C01815=1042.872,189.245,401.631,170.706,39.052,157.377
C01816=1042.879,189.530,401.603,170.709,39.053,157.377
C01817=1042.886,189.814,401.575,170.712,39.055,157.378
C01818=1042.893,190.099,401.548,170.715,39.057,157.378
C01819=1042.899,190.347,401.523,170.718,39.058,157.378
C01820=1042.905,190.596,401.499,170.720,39.060,157.379
C01821=1042.911,190.845,401.475,170.723,39.061,157.379
C01822=1042.918,191.094,401.450,170.726,39.062,157.380
C01823=1042.923,191.342,401.426,170.728,39.064,157.380
C01824=1042.929,191.591,401.402,170.731,39.065,157.380
C01825=1042.935,191.839,401.377,170.734,39.067,157.381
C01826=1042.941,192.089,401.353,170.737,39.068,157.381
C01827=1042.948,192.338,401.329,170.739,39.070,157.381
C01828=1042.953,192.586,401.304,170.742,39.071,157.382
C01829=1042.960,192.835,401.280,170.745,39.072,157.382
C01830=1042.965,193.083,401.255,170.747,39.074,157.383
C01831=1042.972,193.332,401.231,170.750,39.075,157.383
C01832=1042.978,193.581,401.207,170.753,39.077,157.383
C01833=1042.984,193.829,401.182,170.755,39.078,157.384
C01834=1042.990,194.078,401.158,170.759,39.080,157.384
C01835=1042.997,194.327,401.134,170.761,39.081,157.384
C01836=1043.002,194.575,401.109,170.763,39.082,157.385
C01837=1043.009,194.824,401.085,170.767,39.084,157.385
C01838=1043.015,195.074,401.060,170.769,39.085,157.385
C01839=1043.021,195.322,401.035,170.772,39.087,157.386
C01840=1043.027,195.571,401.011,170.775,39.088,157.386
C01841=1043.033,195.819,400.986,170.778,39.089,157.387
C01842=1043.040,196.068,400.962,170.780,39.091,157.387
C01843=1043.045,196.317,400.937,170.783,39.093,157.387
C01844=1043.052,196.565,400.913,170.786,39.094,157.388
C01845=1043.058,196.814,400.888,170.789,39.096,157.388
C01846=1043.064,197.063,400.863,170.792,39.097,157.389
C01847=1043.070,197.311,400.839,170.794,39.098,157.389
C01848=1043.076,197.560,400.814,170.798,39.100,157.389
C01849=1043.083,197.809,400.790,170.800,39.101,157.390
C01850=1043.089,198.058,400.765,170.802,39.103,157.390
C01851=1043.096,198.307,400.740,170.806,39.105,157.391
C01852=1043.101,198.555,400.716,170.808,39.106,157.391
C01853=1043.107,198.804,400.691,170.811,39.107,157.391
C01854=1043.114,199.053,400.667,170.814,39.109,157.392
C01855=1043.120,199.302,400.641,170.817,39.110,157.392
C01856=1043.127,199.550,400.617,170.819,39.112,157.392
C01857=1043.132,199.798,400.592,170.823,39.113,157.393
C01858=1043.139,200.047,400.568,170.825,39.114,157.393
C01859=1043.145,200.296,400.543,170.828,39.116,157.394
C01860=1043.152,200.545,400.518,170.831,39.118,157.394
C01861=1043.158,200.794,400.494,170.834,39.119,157.394
C01862=1043.164,201.042,400.468,170.836,39.121,157.395
C01863=1043.170,201.290,400.443,170.840,39.122,157.395
C01864=1043.176,201.540,400.419,170.842,39.124,157.396
C01865=1043.183,201.788,400.394,170.846,39.126,157.396
C01866=1043.189,202.037,400.369,170.848,39.127,157.396
C01867=1043.195,202.285,400.343,170.850,39.129,157.397
C01868=1043.201,202.535,400.319,170.854,39.130,157.397
C01869=1043.207,202.783,400.294,170.856,39.132,157.398
C01870=1043.213,203.031,400.268,170.860,39.133,157.398
C01871=1043.219,203.280,400.243,170.862,39.135,157.398
C01872=1043.225,203.529,400.218,170.865,39.137,157.399
C01873=1043.231,203.778,400.193,170.868,39.138,157.399
C01874=1043.237,204.027,400.168,170.871,39.140,157.400
C01875=1043.243,204.275,400.143,170.873,39.142,157.400
C01876=1043.249,204.523,400.117,170.877,39.143,157.401
C01877=1043.255,204.772,400.092,170.879,39.145,157.401
C01878=1043.262,205.021,400.068,170.883,39.147,157.401
C01879=1043.288,206.072,399.961,171.152,39.248,157.431
C01880=1043.296,206.361,399.930,171.154,39.251,157.431
C01881=1043.303,206.650,399.900,171.156,39.254,157.432
C01882=1043.311,206.938,399.870,171.159,39.257,157.432
C01883=1043.319,207.228,399.839,171.162,39.260,157.433
C01884=1043.326,207.476,399.813,171.164,39.262,157.434
C01885=1043.332,207.725,399.786,171.166,39.264,157.434
C01886=1043.339,207.973,399.759,171.168,39.267,157.435
C01887=1043.346,208.222,399.733,171.170,39.269,157.435
C01888=1043.352,208.470,399.707,171.172,39.271,157.436
C01889=1043.359,208.719,399.680,171.175,39.273,157.436
C01890=1043.365,208.967,399.654,171.177,39.276,157.437
C01891=1043.372,209.215,399.628,171.179,39.279,157.438
C01892=1043.379,209.465,399.601,171.181,39.281,157.438
C01893=1043.385,209.713,399.574,171.183,39.283,157.439
C01894=1043.392,209.962,399.547,171.186,39.286,157.439
C01895=1043.398,210.210,399.521,171.187,39.288,157.440
C01896=1043.405,210.458,399.495,171.190,39.290,157.440
C01897=1043.411,210.707,399.468,171.191,39.293,157.441
C01898=1043.418,210.956,399.442,171.194,39.295,157.442
C01899=1043.425,211.203,399.415,171.196,39.297,157.442
C01900=1043.431,211.452,399.388,171.198,39.300,157.443
C01901=1043.438,211.701,399.362,171.200,39.302,157.443
C01902=1043.444,211.949,399.335,171.203,39.304,157.444
C01903=1043.451,212.198,399.309,171.205,39.307,157.445
C01904=1043.457,212.446,399.282,171.207,39.310,157.445
C01905=1043.464,212.694,399.255,171.209,39.312,157.446
C01906=1043.470,212.943,399.228,171.211,39.314,157.446
C01907=1043.477,213.192,399.202,171.214,39.317,157.447
C01908=1043.484,213.441,399.175,171.215,39.319,157.447
C01909=1043.490,213.688,399.147,171.218,39.321,157.448
C01910=1043.497,213.937,399.121,171.220,39.324,157.448
C01911=1043.503,214.185,399.094,171.222,39.327,157.449
C01912=1043.510,214.434,399.068,171.225,39.329,157.450
C01913=1043.516,214.683,399.040,171.227,39.331,157.450
C01914=1043.523,214.931,399.014,171.229,39.334,157.451
C01915=1043.529,215.180,398.987,171.231,39.336,157.451
C01916=1043.537,215.428,398.960,171.234,39.338,157.452
C01917=1043.543,215.676,398.933,171.235,39.341,157.452
C01918=1043.549,215.925,398.906,171.238,39.343,157.453
C01919=1043.556,216.173,398.879,171.240,39.345,157.454
C01920=1043.562,216.422,398.853,171.242,39.348,157.454
C01921=1043.569,216.671,398.826,171.244,39.350,157.455
C01922=1043.576,216.919,398.798,171.247,39.352,157.455
C01923=1043.582,217.167,398.772,171.248,39.355,157.456
C01924=1043.589,217.416,398.745,171.251,39.357,157.456
C01925=1043.595,217.665,398.718,171.254,39.360,157.457
C01926=1043.602,217.913,398.692,171.256,39.362,157.458
C01927=1043.609,218.161,398.664,171.258,39.364,157.458
C01928=1043.616,218.410,398.637,171.260,39.367,157.459
C01929=1043.622,218.658,398.611,171.263,39.369,157.459
C01930=1043.628,218.907,398.583,171.264,39.371,157.460
C01931=1043.635,219.155,398.557,171.267,39.374,157.460
C01932=1043.642,219.404,398.529,171.269,39.376,157.461
C01933=1043.649,219.652,398.503,171.272,39.378,157.461
C01934=1043.655,219.900,398.475,171.274,39.381,157.462
C01935=1043.662,220.149,398.448,171.276,39.383,157.463
C01936=1043.670,220.443,398.416,171.279,39.386,157.463
C01937=1043.678,220.737,398.384,171.281,39.389,157.464
C01938=1043.685,221.032,398.351,171.284,39.391,157.465
C01939=1043.692,221.326,398.320,171.287,39.394,157.465
C01940=1043.699,221.574,398.292,171.289,39.396,157.466
C01941=1043.706,221.823,398.264,171.292,39.399,157.467
C01942=1043.712,222.072,398.237,171.293,39.402,157.467
C01943=1043.718,222.320,398.210,171.296,39.404,157.468
C01944=1043.726,222.568,398.183,171.299,39.406,157.468
C01945=1043.732,222.817,398.156,171.301,39.408,157.469
C01946=1043.739,223.065,398.128,171.304,39.411,157.469
C01947=1043.745,223.313,398.101,171.305,39.413,157.470
C01948=1043.751,223.562,398.074,171.308,39.415,157.470
C01949=1043.758,223.810,398.046,171.310,39.418,157.471
C01950=1043.765,224.059,398.018,171.313,39.420,157.472
C01951=1043.771,224.308,397.991,171.314,39.422,157.472
C01952=1043.778,224.555,397.964,171.317,39.425,157.473
C01953=1043.784,224.804,397.937,171.320,39.427,157.473
C01954=1043.791,225.052,397.909,171.322,39.430,157.474
C01955=1043.797,225.301,397.882,171.324,39.432,157.474
C01956=1043.804,225.550,397.854,171.326,39.434,157.475
C01957=1043.810,225.798,397.827,171.329,39.437,157.476
C01958=1043.817,226.046,397.799,171.331,39.439,157.476
C01959=1043.824,226.294,397.771,171.334,39.441,157.477
C01960=1043.831,226.543,397.745,171.336,39.444,157.477
C01961=1043.837,226.792,397.717,171.338,39.446,157.478
C01962=1043.844,227.040,397.689,171.340,39.448,157.478
C01963=1043.851,227.288,397.662,171.343,39.450,157.479
C01964=1043.857,227.536,397.634,171.346,39.453,157.480
C01965=1043.864,227.785,397.607,171.348,39.455,157.480
C01966=1043.870,228.034,397.580,171.350,39.457,157.481
C01967=1043.877,228.282,397.552,171.352,39.460,157.481
C01968=1043.883,228.531,397.524,171.355,39.462,157.482
C01969=1043.890,228.779,397.496,171.357,39.464,157.482
C01970=1043.897,229.027,397.469,171.360,39.467,157.483
C01971=1043.903,229.276,397.441,171.363,39.469,157.484
C01972=1043.909,229.524,397.414,171.364,39.472,157.484
C01973=1043.916,229.772,397.386,171.367,39.474,157.485
C01974=1043.923,230.021,397.358,171.369,39.476,157.485
C01975=1043.929,230.269,397.330,171.372,39.479,157.486
C01976=1043.936,230.517,397.303,171.374,39.481,157.486
C01977=1043.943,230.766,397.275,171.377,39.483,157.487
C01978=1043.949,231.015,397.247,171.379,39.485,157.488
C01979=1043.955,231.263,397.219,171.381,39.488,157.488
C01980=1043.962,231.512,397.191,171.384,39.491,157.489
C01981=1043.968,231.759,397.164,171.386,39.493,157.489
C01982=1043.975,232.008,397.136,171.389,39.495,157.490
C01983=1043.982,232.255,397.108,171.391,39.498,157.491
C01984=1043.989,232.504,397.080,171.394,39.500,157.491
C01985=1043.994,232.753,397.052,171.396,39.502,157.492
C01986=1044.001,233.001,397.024,171.398,39.504,157.492
C01987=1044.008,233.250,396.996,171.401,39.507,157.493
C01988=1044.015,233.498,396.968,171.403,39.510,157.494
C01989=1044.020,233.747,396.940,171.406,39.512,157.494
C01990=1044.027,233.995,396.912,171.408,39.514,157.495
C01991=1044.034,234.243,396.884,171.411,39.516,157.495
C01992=1044.041,234.530,396.852,171.414,39.519,157.496
C01993=1044.049,234.817,396.819,171.416,39.522,157.496
C01994=1044.056,235.103,396.787,171.419,39.525,157.497
C01995=1044.064,235.390,396.754,171.423,39.527,157.498
C01996=1044.071,235.639,396.727,171.424,39.530,157.498
C01997=1044.077,235.887,396.698,171.427,39.532,157.499
C01998=1044.084,236.135,396.670,171.429,39.534,157.500
C01999=1044.090,236.384,396.642,171.432,39.537,157.500
C02000=1044.096,236.632,396.614,171.434,39.539,157.501
C02001=1044.103,236.880,396.585,171.437,39.542,157.501
C02002=1044.110,237.129,396.558,171.440,39.544,157.502
C02003=1044.117,237.377,396.530,171.442,39.546,157.503
C02004=1044.123,237.625,396.501,171.445,39.548,157.503
C02005=1044.130,237.874,396.473,171.447,39.551,157.504
C02006=1044.137,238.122,396.445,171.450,39.553,157.504
C02007=1044.143,238.370,396.416,171.452,39.555,157.505
C02008=1044.149,238.619,396.389,171.455,39.558,157.505
C02009=1044.156,238.867,396.360,171.458,39.560,157.506
C02010=1044.162,239.115,396.332,171.460,39.563,157.507
C02011=1044.169,239.363,396.304,171.463,39.565,157.507
C02012=1044.176,239.612,396.276,171.465,39.567,157.508
C02013=1044.183,239.860,396.246,171.467,39.570,157.508
C02014=1044.189,240.109,396.219,171.469,39.572,157.509
C02015=1044.195,240.358,396.190,171.472,39.574,157.510
C02016=1044.202,240.605,396.162,171.475,39.576,157.510
C02017=1044.209,240.854,396.134,171.477,39.579,157.511
C02018=1044.215,241.102,396.105,171.480,39.581,157.511
C02019=1044.222,241.350,396.077,171.482,39.583,157.512
C02020=1044.228,241.599,396.048,171.485,39.586,157.513
C02021=1044.235,241.846,396.020,171.488,39.588,157.513
C02022=1044.241,242.095,395.992,171.490,39.591,157.514
C02023=1044.248,242.343,395.963,171.493,39.593,157.514
C02024=1044.255,242.592,395.934,171.495,39.595,157.515
C02025=1044.261,242.841,395.905,171.498,39.598,157.516
C02026=1044.268,243.088,395.877,171.501,39.600,157.516
C02027=1044.274,243.336,395.848,171.503,39.603,157.517
C02028=1044.281,243.585,395.820,171.506,39.605,157.517
C02029=1044.287,243.833,395.791,171.508,39.607,157.518
C02030=1044.293,244.081,395.762,171.511,39.610,157.519
C02031=1044.300,244.330,395.734,171.513,39.612,157.519
C02032=1044.307,244.578,395.705,171.516,39.615,157.520
C02033=1044.314,244.826,395.677,171.519,39.617,157.520
C02034=1044.320,245.074,395.647,171.521,39.619,157.521
C02035=1044.326,245.323,395.619,171.524,39.621,157.521
C02036=1044.333,245.571,395.591,171.526,39.624,157.522
C02037=1044.339,245.819,395.562,171.529,39.626,157.523
C02038=1044.346,246.067,395.533,171.532,39.629,157.523
C02039=1044.352,246.315,395.504,171.534,39.632,157.524
C02040=1044.359,246.564,395.474,171.537,39.634,157.525
C02041=1044.365,246.813,395.446,171.539,39.636,157.525
C02042=1044.371,247.061,395.417,171.542,39.638,157.526
C02043=1044.378,247.309,395.388,171.545,39.641,157.526
C02044=1044.384,247.557,395.359,171.547,39.643,157.527
C02045=1044.390,247.805,395.330,171.551,39.646,157.528
C02046=1044.397,248.054,395.301,171.553,39.648,157.528
C02047=1044.403,248.302,395.272,171.556,39.651,157.529
C02048=1044.410,248.583,395.239,171.559,39.654,157.530
C02049=1044.418,248.864,395.206,171.561,39.656,157.530
C02050=1044.426,249.145,395.174,171.565,39.659,157.531
C02051=1044.433,249.425,395.141,171.568,39.662,157.532
C02052=1044.440,249.674,395.111,171.570,39.664,157.532
C02053=1044.446,249.922,395.082,171.573,39.667,157.533
C02054=1044.452,250.170,395.053,171.576,39.669,157.533
C02055=1044.458,250.419,395.024,171.578,39.671,157.534
C02056=1044.465,250.667,394.995,171.581,39.673,157.535
C02057=1044.471,250.916,394.966,171.584,39.676,157.535
C02058=1044.478,251.163,394.937,171.586,39.679,157.536
C02059=1044.485,251.411,394.908,171.590,39.681,157.536
C02060=1044.491,251.660,394.879,171.592,39.683,157.537
C02061=1044.498,251.908,394.850,171.595,39.686,157.538
C02062=1044.504,252.157,394.821,171.598,39.688,157.538
C02063=1044.511,252.404,394.791,171.600,39.690,157.539
C02064=1044.517,252.653,394.762,171.603,39.693,157.539
C02065=1044.524,252.901,394.733,171.605,39.695,157.540
C02066=1044.530,253.149,394.704,171.608,39.698,157.541
C02067=1044.537,253.398,394.674,171.611,39.700,157.541
C02068=1044.544,253.646,394.646,171.614,39.702,157.542
C02069=1044.550,253.893,394.616,171.617,39.705,157.543
C02070=1044.557,254.142,394.587,171.619,39.707,157.543
C02071=1044.563,254.390,394.557,171.622,39.709,157.544
C02072=1044.570,254.638,394.528,171.625,39.712,157.544
C02073=1044.577,254.887,394.498,171.627,39.715,157.545
C02074=1044.583,255.135,394.469,171.630,39.717,157.546
C02075=1044.589,255.383,394.440,171.633,39.719,157.546
C02076=1044.596,255.632,394.411,171.636,39.721,157.547
C02077=1044.603,255.879,394.381,171.639,39.724,157.547
C02078=1044.610,256.128,394.352,171.641,39.726,157.548
C02079=1044.616,256.376,394.323,171.644,39.729,157.549
C02080=1044.623,256.623,394.293,171.647,39.731,157.549
C02081=1044.630,256.872,394.264,171.650,39.733,157.550
C02082=1044.636,257.120,394.235,171.653,39.736,157.551
C02083=1044.643,257.369,394.205,171.655,39.738,157.551
C02084=1044.650,257.617,394.176,171.658,39.740,157.552
C02085=1044.656,257.864,394.146,171.661,39.743,157.552
C02086=1044.663,258.113,394.117,171.664,39.745,157.553
C02087=1044.669,258.361,394.088,171.667,39.748,157.554
C02088=1044.676,258.609,394.058,171.669,39.750,157.554
C02089=1044.683,258.858,394.029,171.672,39.752,157.555
C02090=1044.690,259.106,393.998,171.676,39.755,157.556
C02091=1044.696,259.354,393.969,171.678,39.757,157.556
C02092=1044.703,259.602,393.939,171.681,39.759,157.557
C02093=1044.709,259.850,393.910,171.683,39.762,157.557
C02094=1044.717,260.098,393.880,171.686,39.764,157.558
C02095=1044.723,260.347,393.851,171.690,39.767,157.559
C02096=1044.730,260.595,393.821,171.692,39.769,157.559
C02097=1044.736,260.843,393.792,171.695,39.771,157.560
C02098=1044.743,261.091,393.762,171.698,39.773,157.560
C02099=1044.750,261.339,393.733,171.701,39.776,157.561
C02100=1044.757,261.588,393.703,171.704,39.778,157.562
C02101=1044.763,261.836,393.674,171.706,39.781,157.562
C02102=1044.771,262.084,393.644,171.709,39.783,157.563
C02103=1044.778,262.332,393.614,171.713,39.785,157.563
C02104=1044.785,262.611,393.581,171.715,39.788,157.564
C02105=1044.792,262.891,393.547,171.719,39.791,157.565
C02106=1044.800,263.171,393.513,171.722,39.793,157.566
C02107=1044.806,263.450,393.480,171.726,39.796,157.566
C02108=1044.814,263.698,393.450,171.728,39.799,157.567
C02109=1044.819,263.946,393.419,171.731,39.801,157.568
C02110=1044.827,264.194,393.389,171.734,39.803,157.568
C02111=1044.833,264.442,393.359,171.737,39.806,157.569
C02112=1044.839,264.691,393.329,171.740,39.808,157.569
C02113=1044.846,264.939,393.299,171.742,39.811,157.570
C02114=1044.853,265.187,393.269,171.746,39.813,157.571
C02115=1044.859,265.435,393.239,171.749,39.816,157.571
C02116=1044.866,265.683,393.209,171.751,39.819,157.572
C02117=1044.873,265.931,393.179,171.755,39.821,157.573
C02118=1044.879,266.179,393.149,171.758,39.824,157.573
C02119=1044.886,266.428,393.119,171.760,39.826,157.574
C02120=1044.893,266.676,393.089,171.763,39.828,157.575
C02121=1044.899,266.924,393.059,171.767,39.831,157.575
C02122=1044.906,267.172,393.029,171.769,39.833,157.576
C02123=1044.912,267.419,392.999,171.772,39.836,157.577
C02124=1044.919,267.668,392.968,171.776,39.838,157.577
C02125=1044.926,267.916,392.938,171.778,39.841,157.578
C02126=1044.932,268.164,392.908,171.781,39.843,157.579
C02127=1044.939,268.412,392.877,171.784,39.845,157.579
C02128=1044.945,268.660,392.847,171.787,39.848,157.580
C02129=1044.952,268.908,392.817,171.790,39.850,157.580
C02130=1044.958,269.157,392.786,171.794,39.853,157.581
C02131=1044.965,269.404,392.757,171.796,39.855,157.582
C02132=1044.971,269.653,392.726,171.799,39.858,157.582
C02133=1044.979,269.900,392.695,171.802,39.860,157.583
C02134=1044.985,270.148,392.665,171.805,39.863,157.584
C02135=1044.992,270.396,392.634,171.808,39.865,157.584
C02136=1044.998,270.645,392.604,171.811,39.868,157.585
C02137=1045.005,270.892,392.574,171.814,39.870,157.586
C02138=1045.011,271.141,392.543,171.817,39.873,157.586
C02139=1045.018,271.389,392.513,171.820,39.875,157.587
C02140=1045.024,271.636,392.482,171.823,39.878,157.588
C02141=1045.032,271.884,392.452,171.826,39.880,157.588
C02142=1045.038,272.133,392.421,171.829,39.883,157.589
C02143=1045.044,272.381,392.391,171.832,39.885,157.590
C02144=1045.051,272.628,392.360,171.836,39.888,157.590
C02145=1045.058,272.877,392.329,171.838,39.890,157.591
C02146=1045.063,273.125,392.299,171.841,39.893,157.592
C02147=1045.071,273.373,392.269,171.845,39.895,157.592
C02148=1045.077,273.621,392.237,171.847,39.898,157.593
C02149=1045.084,273.869,392.207,171.850,39.900,157.594
C02150=1045.091,274.116,392.176,171.854,39.903,157.594
C02151=1045.097,274.365,392.146,171.857,39.906,157.595
C02152=1045.103,274.613,392.115,171.860,39.908,157.596
C02153=1045.111,274.861,392.084,171.863,39.911,157.596
C02154=1045.117,275.109,392.054,171.866,39.913,157.597
C02155=1045.123,275.357,392.022,171.869,39.916,157.598
C02156=1045.130,275.605,391.992,171.872,39.918,157.598
C02157=1045.137,275.853,391.961,171.876,39.921,157.599
C02158=1045.143,276.101,391.930,171.878,39.923,157.600
C02159=1045.150,276.349,391.900,171.882,39.926,157.600
C02160=1045.158,276.633,391.864,171.885,39.928,157.601
C02161=1045.165,276.917,391.829,171.889,39.932,157.602
C02162=1045.173,277.201,391.793,171.892,39.934,157.603
C02163=1045.181,277.485,391.758,171.896,39.937,157.603
C02164=1045.187,277.732,391.727,171.899,39.940,157.604
C02165=1045.193,277.981,391.696,171.902,39.942,157.605
C02166=1045.200,278.229,391.665,171.905,39.945,157.606
C02167=1045.207,278.476,391.634,171.908,39.948,157.606
C02168=1045.214,278.725,391.603,171.912,39.950,157.607
C02169=1045.220,278.973,391.572,171.914,39.953,157.608
C02170=1045.227,279.221,391.541,171.918,39.955,157.608
C02171=1045.233,279.468,391.510,171.921,39.958,157.609
C02172=1045.240,279.716,391.479,171.924,39.960,157.610
C02173=1045.246,279.964,391.447,171.927,39.963,157.610
C02174=1045.253,280.213,391.416,171.931,39.965,157.611
C02175=1045.260,280.461,391.385,171.933,39.968,157.612
C02176=1045.266,280.709,391.354,171.937,39.971,157.612
C02177=1045.272,280.956,391.323,171.940,39.974,157.613
C02178=1045.279,281.204,391.292,171.944,39.976,157.614
C02179=1045.286,281.452,391.260,171.946,39.979,157.614
C02180=1045.292,281.700,391.229,171.950,39.981,157.615
C02181=1045.299,281.948,391.198,171.953,39.984,157.616
C02182=1045.306,282.196,391.166,171.956,39.986,157.617
C02183=1045.312,282.444,391.135,171.959,39.989,157.617
C02184=1045.319,282.692,391.103,171.963,39.992,157.618
C02185=1045.326,282.940,391.072,171.966,39.995,157.619
C02186=1045.332,283.187,391.041,171.969,39.997,157.619
C02187=1045.338,283.435,391.010,171.972,40.000,157.620
C02188=1045.345,283.683,390.979,171.976,40.002,157.621
C02189=1045.352,283.931,390.947,171.979,40.005,157.622
C02190=1045.359,284.179,390.916,171.982,40.007,157.622
C02191=1045.365,284.427,390.884,171.985,40.010,157.623
C02192=1045.372,284.675,390.853,171.989,40.013,157.624
C02193=1045.379,284.923,390.821,171.991,40.016,157.624
C02194=1045.386,285.171,390.790,171.995,40.018,157.625
C02195=1045.392,285.419,390.759,171.998,40.020,157.626
C02196=1045.399,285.666,390.727,172.002,40.023,157.626
C02197=1045.406,285.914,390.696,172.005,40.026,157.627
C02198=1045.412,286.162,390.664,172.008,40.028,157.628
C02199=1045.419,286.410,390.633,172.012,40.031,157.629
C02200=1045.426,286.658,390.601,172.014,40.034,157.629
C02201=1045.432,286.906,390.569,172.018,40.036,157.630
C02202=1045.439,287.154,390.537,172.021,40.039,157.631
C02203=1045.446,287.401,390.506,172.025,40.041,157.631
C02204=1045.452,287.649,390.474,172.028,40.044,157.632
C02205=1045.460,287.898,390.443,172.031,40.047,157.633
C02206=1045.466,288.146,390.411,172.035,40.049,157.634
C02207=1045.473,288.393,390.378,172.038,40.052,157.634
C02208=1045.479,288.641,390.347,172.041,40.055,157.635
C02209=1045.486,288.889,390.315,172.045,40.058,157.636
C02210=1045.493,289.137,390.284,172.048,40.060,157.637
C02211=1045.499,289.385,390.251,172.052,40.063,157.637
C02212=1045.506,289.633,390.220,172.054,40.065,157.638
C02213=1045.513,289.881,390.188,172.058,40.068,157.639
C02214=1045.520,290.128,390.156,172.062,40.071,157.639
C02215=1045.526,290.376,390.124,172.065,40.074,157.640
C02216=1045.534,290.672,390.086,172.069,40.077,157.641
C02217=1045.542,290.967,390.048,172.072,40.080,157.642
C02218=1045.550,291.263,390.010,172.077,40.083,157.643
C02219=1045.558,291.559,389.972,172.081,40.087,157.644
C02220=1045.564,291.806,389.939,172.084,40.089,157.644
C02221=1045.571,292.054,389.908,172.088,40.092,157.645
C02222=1045.578,292.302,389.876,172.092,40.095,157.646
C02223=1045.584,292.550,389.844,172.094,40.098,157.647
C02224=1045.591,292.798,389.812,172.098,40.100,157.647
C02225=1045.599,293.045,389.780,172.102,40.103,157.648
C02226=1045.605,293.293,389.747,172.105,40.106,157.649
C02227=1045.612,293.541,389.715,172.108,40.109,157.650
C02228=1045.618,293.789,389.683,172.112,40.111,157.650
C02229=1045.625,294.036,389.651,172.115,40.114,157.651
C02230=1045.632,294.284,389.619,172.119,40.117,157.652
C02231=1045.638,294.532,389.586,172.123,40.119,157.653
C02232=1045.645,294.780,389.555,172.125,40.122,157.653
C02233=1045.651,295.028,389.522,172.129,40.125,157.654
C02234=1045.659,295.275,389.490,172.133,40.128,157.655
C02235=1045.665,295.524,389.457,172.136,40.130,157.656
C02236=1045.672,295.771,389.425,172.139,40.133,157.656
C02237=1045.678,296.019,389.392,172.143,40.136,157.657
C02238=1045.685,296.266,389.360,172.147,40.138,157.658
C02239=1045.691,296.515,389.327,172.150,40.142,157.659
C02240=1045.698,296.762,389.295,172.154,40.145,157.660
C02241=1045.705,297.010,389.262,172.157,40.147,157.660
C02242=1045.711,297.258,389.230,172.160,40.150,157.661
C02243=1045.717,297.505,389.197,172.164,40.153,157.662
C02244=1045.724,297.752,389.165,172.168,40.156,157.663
C02245=1045.731,298.001,389.132,172.171,40.159,157.663
C02246=1045.737,298.248,389.099,172.174,40.161,157.664
C02247=1045.744,298.496,389.066,172.178,40.165,157.665
C02248=1045.750,298.744,389.034,172.181,40.168,157.666
C02249=1045.757,298.992,389.002,172.185,40.170,157.667
C02250=1045.764,299.240,388.969,172.189,40.173,157.667
C02251=1045.770,299.487,388.936,172.193,40.176,157.668
C02252=1045.777,299.736,388.903,172.195,40.179,157.669
C02253=1045.783,299.983,388.870,172.199,40.182,157.670
C02254=1045.790,300.230,388.837,172.203,40.184,157.670
C02255=1045.797,300.477,388.805,172.207,40.188,157.671
C02256=1045.804,300.726,388.772,172.210,40.190,157.672
C02257=1045.810,300.973,388.739,172.213,40.193,157.673
C02258=1045.816,301.221,388.706,172.217,40.196,157.674
C02259=1045.824,301.469,388.674,172.221,40.199,157.674
C02260=1045.830,301.716,388.641,172.224,40.202,157.675
C02261=1045.836,301.964,388.608,172.228,40.205,157.676
C02262=1045.844,302.212,388.574,172.232,40.208,157.677
C02263=1045.850,302.459,388.541,172.235,40.210,157.678
C02264=1045.857,302.708,388.508,172.239,40.214,157.679
C02265=1045.864,302.955,388.476,172.242,40.216,157.679
C02266=1045.870,303.203,388.443,172.246,40.219,157.680
C02267=1045.877,303.450,388.410,172.250,40.222,157.681
C02268=1045.884,303.698,388.377,172.254,40.225,157.682
C02269=1045.891,303.946,388.344,172.257,40.228,157.682
C02270=1045.897,304.194,388.311,172.261,40.231,157.683
C02271=1045.904,304.441,388.277,172.264,40.234,157.684
C02272=1045.913,304.753,388.237,172.269,40.238,157.685
C02273=1045.921,305.065,388.195,172.273,40.241,157.686
C02274=1045.930,305.377,388.153,172.278,40.245,157.687
C02275=1045.939,305.688,388.111,172.283,40.248,157.688
C02276=1045.945,305.937,388.078,172.287,40.252,157.689
C02277=1045.952,306.184,388.045,172.290,40.254,157.690
C02278=1045.959,306.432,388.012,172.294,40.257,157.691
C02279=1045.965,306.679,387.979,172.298,40.260,157.691
C02280=1045.972,306.927,387.945,172.302,40.263,157.692
C02281=1045.979,307.174,387.913,172.306,40.266,157.693
C02282=1045.987,307.422,387.879,172.309,40.269,157.694
C02283=1045.993,307.670,387.846,172.313,40.272,157.695
C02284=1046.000,307.917,387.812,172.317,40.275,157.696
C02285=1046.007,308.166,387.779,172.320,40.278,157.696
C02286=1046.014,308.413,387.746,172.324,40.281,157.697
C02287=1046.020,308.661,387.713,172.328,40.284,157.698
C02288=1046.027,308.908,387.679,172.332,40.287,157.699
C02289=1046.034,309.155,387.645,172.335,40.289,157.700
C02290=1046.042,309.403,387.613,172.339,40.293,157.700
C02291=1046.049,309.650,387.579,172.343,40.295,157.701
C02292=1046.055,309.899,387.546,172.347,40.299,157.702
C02293=1046.063,310.146,387.513,172.351,40.301,157.703
C02294=1046.069,310.393,387.479,172.355,40.305,157.704
C02295=1046.076,310.642,387.446,172.359,40.307,157.705
C02296=1046.083,310.889,387.412,172.363,40.310,157.705
C02297=1046.090,311.136,387.379,172.366,40.313,157.706
C02298=1046.097,311.384,387.345,172.370,40.316,157.707
C02299=1046.104,311.632,387.312,172.374,40.319,157.708
C02300=1046.111,311.880,387.278,172.378,40.322,157.709
C02301=1046.119,312.127,387.245,172.382,40.325,157.710
C02302=1046.126,312.374,387.211,172.386,40.328,157.711
C02303=1046.133,312.623,387.178,172.390,40.331,157.711
C02304=1046.139,312.870,387.144,172.393,40.334,157.712
C02305=1046.146,313.118,387.110,172.397,40.337,157.713
C02306=1046.152,313.366,387.076,172.401,40.341,157.714
C02307=1046.159,313.613,387.042,172.404,40.344,157.715
C02308=1046.165,313.861,387.008,172.408,40.347,157.716
C02309=1046.172,314.108,386.974,172.412,40.350,157.717
C02310=1046.178,314.355,386.940,172.416,40.353,157.717
C02311=1046.185,314.603,386.906,172.420,40.356,157.718
C02312=1046.193,314.850,386.872,172.424,40.360,157.719
C02313=1046.199,315.097,386.838,172.428,40.363,157.720
C02314=1046.206,315.345,386.804,172.432,40.366,157.721
C02315=1046.213,315.593,386.769,172.436,40.369,157.722
C02316=1046.220,315.841,386.736,172.440,40.372,157.723
C02317=1046.226,316.088,386.702,172.444,40.376,157.724
C02318=1046.233,316.336,386.668,172.448,40.378,157.725
C02319=1046.240,316.583,386.633,172.452,40.382,157.725
C02320=1046.247,316.831,386.599,172.456,40.385,157.726
C02321=1046.253,317.079,386.564,172.460,40.388,157.727
C02322=1046.260,317.326,386.531,172.464,40.391,157.728
C02323=1046.267,317.573,386.496,172.468,40.395,157.729
C02324=1046.274,317.821,386.462,172.471,40.398,157.730
C02325=1046.280,318.069,386.427,172.475,40.401,157.731
C02326=1046.287,318.316,386.394,172.479,40.404,157.732
C02327=1046.294,318.564,386.359,172.483,40.407,157.733
C02328=1046.302,318.880,386.315,172.489,40.412,157.734
C02329=1046.312,319.197,386.271,172.494,40.415,157.735
C02330=1046.320,319.513,386.227,172.499,40.420,157.736
C02331=1046.329,319.829,386.183,172.504,40.424,157.737
C02332=1046.336,320.077,386.149,172.508,40.427,157.738
C02333=1046.343,320.324,386.114,172.512,40.431,157.739
C02334=1046.350,320.572,386.080,172.516,40.434,157.740
C02335=1046.357,320.819,386.045,172.520,40.437,157.741
C02336=1046.364,321.067,386.011,172.524,40.440,157.742
C02337=1046.370,321.315,385.976,172.528,40.443,157.743
C02338=1046.378,321.563,385.942,172.532,40.447,157.744
C02339=1046.384,321.810,385.907,172.536,40.450,157.745
C02340=1046.392,322.058,385.873,172.541,40.453,157.746
C02341=1046.398,322.305,385.838,172.545,40.456,157.747
C02342=1046.406,322.552,385.803,172.549,40.459,157.748
C02343=1046.412,322.800,385.769,172.553,40.463,157.748
C02344=1046.419,323.047,385.734,172.557,40.466,157.749
C02345=1046.426,323.295,385.700,172.561,40.470,157.750
C02346=1046.433,323.542,385.665,172.565,40.473,157.751
C02347=1046.440,323.789,385.630,172.569,40.476,157.752
C02348=1046.447,324.037,385.596,172.574,40.479,157.753
C02349=1046.454,324.284,385.561,172.578,40.482,157.754
C02350=1046.461,324.532,385.526,172.582,40.486,157.755
C02351=1046.468,324.779,385.491,172.586,40.489,157.756
C02352=1046.475,325.027,385.457,172.590,40.493,157.757
C02353=1046.482,325.274,385.422,172.594,40.496,157.758
C02354=1046.490,325.522,385.387,172.599,40.499,157.759
C02355=1046.497,325.769,385.352,172.603,40.502,157.760
C02356=1046.504,326.017,385.317,172.607,40.506,157.761
C02357=1046.511,326.264,385.283,172.611,40.509,157.762
C02358=1046.518,326.512,385.248,172.615,40.512,157.763
C02359=1046.525,326.759,385.213,172.620,40.516,157.764
C02360=1046.532,327.007,385.178,172.624,40.519,157.765
C02361=1046.539,327.254,385.143,172.628,40.523,157.766
C02362=1046.547,327.501,385.108,172.632,40.526,157.766
C02363=1046.554,327.749,385.073,172.637,40.529,157.767
C02364=1046.561,327.997,385.038,172.641,40.533,157.768
C02365=1046.568,328.244,385.003,172.645,40.536,157.769
C02366=1046.575,328.491,384.968,172.649,40.539,157.770
C02367=1046.583,328.738,384.933,172.655,40.543,157.771
C02368=1046.590,328.986,384.898,172.658,40.546,157.772
C02369=1046.597,329.234,384.863,172.662,40.549,157.773
C02370=1046.604,329.481,384.828,172.667,40.553,157.774
C02371=1046.612,329.729,384.793,172.672,40.556,157.775
C02372=1046.618,329.976,384.758,172.676,40.560,157.776
C02373=1046.624,330.224,384.722,172.680,40.563,157.777
C02374=1046.632,330.471,384.686,172.684,40.567,157.778
C02375=1046.639,330.719,384.651,172.689,40.570,157.779
C02376=1046.646,330.966,384.615,172.693,40.574,157.780
C02377=1046.652,331.213,384.580,172.697,40.577,157.781
C02378=1046.660,331.460,384.544,172.701,40.581,157.782
C02379=1046.667,331.708,384.509,172.706,40.584,157.783
C02380=1046.674,331.955,384.474,172.711,40.588,157.784
C02381=1046.681,332.202,384.438,172.715,40.591,157.785
C02382=1046.688,332.450,384.402,172.719,40.595,157.786
C02383=1046.695,332.697,384.367,172.724,40.599,157.787
C02384=1046.705,333.009,384.322,172.729,40.603,157.789
C02385=1046.713,333.321,384.277,172.734,40.607,157.790
C02386=1046.722,333.632,384.232,172.740,40.612,157.791
C02387=1046.731,333.943,384.187,172.745,40.616,157.793
C02388=1046.738,334.190,384.151,172.750,40.620,157.794
C02389=1046.745,334.438,384.116,172.755,40.624,157.795
C02390=1046.752,334.685,384.080,172.759,40.627,157.796
C02391=1046.759,334.933,384.045,172.764,40.631,157.797
C02392=1046.766,335.180,384.009,172.768,40.634,157.798
C02393=1046.774,335.428,383.973,172.772,40.638,157.799
C02394=1046.781,335.675,383.937,172.777,40.641,157.800
C02395=1046.789,335.922,383.901,172.781,40.645,157.801
C02396=1046.795,336.169,383.866,172.786,40.649,157.802
C02397=1046.802,336.417,383.829,172.791,40.652,157.803
C02398=1046.809,336.664,383.793,172.795,40.656,157.804
C02399=1046.816,336.911,383.758,172.800,40.660,157.805
C02400=1046.823,337.159,383.721,172.804,40.664,157.806
C02401=1046.830,337.406,383.686,172.808,40.667,157.807
C02402=1046.838,337.653,383.649,172.813,40.671,157.808
C02403=1046.844,337.900,383.613,172.818,40.675,157.809
C02404=1046.852,338.148,383.577,172.823,40.678,157.811
C02405=1046.860,338.395,383.541,172.827,40.682,157.812
C02406=1046.866,338.643,383.505,172.831,40.686,157.813
C02407=1046.873,338.890,383.469,172.836,40.690,157.814
C02408=1046.880,339.137,383.433,172.840,40.693,157.815
C02409=1046.888,339.384,383.397,172.846,40.697,157.816
C02410=1046.894,339.632,383.360,172.850,40.701,157.817
C02411=1046.902,339.879,383.324,172.855,40.704,157.818
C02412=1046.910,340.126,383.288,172.859,40.708,157.819
C02413=1046.916,340.373,383.251,172.863,40.712,157.820
C02414=1046.924,340.621,383.215,172.869,40.716,157.821
C02415=1046.931,340.868,383.179,172.873,40.720,157.823
C02416=1046.938,341.115,383.142,172.878,40.724,157.824
C02417=1046.946,341.362,383.105,172.882,40.727,157.825
C02418=1046.953,341.609,383.070,172.887,40.731,157.826
C02419=1046.960,341.857,383.033,172.892,40.735,157.827
C02420=1046.967,342.104,382.997,172.897,40.738,157.828
C02421=1046.974,342.352,382.960,172.901,40.743,157.829
C02422=1046.981,342.599,382.924,172.906,40.746,157.830
C02423=1046.989,342.846,382.886,172.911,40.750,157.831
C02424=1046.996,343.093,382.850,172.916,40.754,157.833
C02425=1047.003,343.340,382.814,172.920,40.758,157.834
C02426=1047.011,343.587,382.777,172.925,40.762,157.835
C02427=1047.018,343.835,382.740,172.930,40.766,157.836
C02428=1047.025,344.082,382.704,172.935,40.770,157.837
C02429=1047.032,344.329,382.667,172.939,40.773,157.838
C02430=1047.039,344.577,382.630,172.944,40.777,157.840
C02431=1047.047,344.823,382.593,172.949,40.781,157.841
C02432=1047.053,345.070,382.556,172.954,40.785,157.842
C02433=1047.061,345.317,382.519,172.958,40.789,157.843
C02434=1047.068,345.565,382.483,172.963,40.793,157.844
C02435=1047.075,345.812,382.445,172.968,40.797,157.845
C02436=1047.083,346.060,382.409,172.973,40.801,157.846
C02437=1047.090,346.306,382.372,172.978,40.805,157.848
C02438=1047.097,346.554,382.335,172.983,40.809,157.849
C02439=1047.105,346.801,382.298,172.988,40.813,157.850
C02440=1047.113,347.108,382.252,172.993,40.818,157.851
C02441=1047.123,347.417,382.206,173.000,40.823,157.853
C02442=1047.131,347.724,382.159,173.006,40.828,157.854
C02443=1047.140,348.031,382.113,173.012,40.833,157.856
C02444=1047.148,348.278,382.076,173.017,40.837,157.857
C02445=1047.155,348.526,382.039,173.022,40.841,157.858
C02446=1047.162,348.773,382.002,173.027,40.845,157.859
C02447=1047.170,349.020,381.964,173.032,40.849,157.861
C02448=1047.178,349.267,381.927,173.037,40.853,157.862
C02449=1047.185,349.514,381.890,173.041,40.857,157.863
C02450=1047.192,349.761,381.852,173.046,40.861,157.864
C02451=1047.200,350.009,381.816,173.052,40.866,157.865
C02452=1047.207,350.256,381.779,173.056,40.870,157.867
C02453=1047.214,350.503,381.741,173.061,40.873,157.868
C02454=1047.222,350.750,381.704,173.067,40.878,157.869
C02455=1047.229,350.997,381.666,173.071,40.882,157.870
C02456=1047.236,351.244,381.629,173.077,40.886,157.872
C02457=1047.243,351.491,381.591,173.082,40.890,157.873
C02458=1047.251,351.738,381.554,173.086,40.895,157.874
C02459=1047.259,351.985,381.517,173.092,40.899,157.875
C02460=1047.266,352.232,381.478,173.097,40.903,157.877
C02461=1047.273,352.479,381.441,173.101,40.907,157.878
C02462=1047.281,352.726,381.403,173.107,40.911,157.879
C02463=1047.288,352.973,381.366,173.112,40.916,157.880
C02464=1047.295,353.220,381.328,173.118,40.920,157.882
C02465=1047.303,353.467,381.290,173.122,40.924,157.883
C02466=1047.310,353.714,381.252,173.127,40.928,157.884
C02467=1047.318,353.962,381.215,173.133,40.932,157.885
C02468=1047.325,354.209,381.177,173.138,40.936,157.887
C02469=1047.332,354.455,381.139,173.143,40.941,157.888
C02470=1047.340,354.703,381.101,173.148,40.946,157.889
C02471=1047.347,354.950,381.064,173.153,40.950,157.890
C02472=1047.355,355.196,381.026,173.159,40.954,157.892
C02473=1047.362,355.443,380.988,173.163,40.958,157.893
C02474=1047.370,355.691,380.949,173.169,40.962,157.894
C02475=1047.377,355.938,380.912,173.174,40.967,157.896
C02476=1047.385,356.184,380.874,173.180,40.971,157.897
C02477=1047.392,356.431,380.836,173.185,40.975,157.898
C02478=1047.400,356.678,380.798,173.189,40.980,157.899
C02479=1047.407,356.926,380.760,173.195,40.984,157.901
C02480=1047.415,357.172,380.722,173.200,40.988,157.902
C02481=1047.422,357.419,380.684,173.206,40.993,157.903
C02482=1047.430,357.666,380.646,173.211,40.997,157.905
C02483=1047.437,357.913,380.607,173.216,41.002,157.906
C02484=1047.444,358.161,380.569,173.221,41.006,157.907
C02485=1047.452,358.407,380.531,173.227,41.010,157.909
C02486=1047.460,358.654,380.492,173.232,41.015,157.910
C02487=1047.467,358.901,380.455,173.238,41.019,157.911
C02488=1047.474,359.148,380.416,173.243,41.024,157.913
C02489=1047.482,359.395,380.377,173.248,41.028,157.914
C02490=1047.490,359.642,380.339,173.253,41.033,157.915
C02491=1047.497,359.889,380.301,173.259,41.037,157.917
C02492=1047.506,360.136,380.262,173.264,41.042,157.918
C02493=1047.512,360.383,380.223,173.270,41.046,157.919
C02494=1047.520,360.630,380.186,173.275,41.051,157.921
C02495=1047.528,360.877,380.147,173.281,41.055,157.922
C02496=1047.537,361.189,380.098,173.288,41.061,157.924
C02497=1047.547,361.503,380.049,173.295,41.067,157.926
C02498=1047.557,361.816,380.000,173.302,41.073,157.927
C02499=1047.566,362.129,379.952,173.309,41.078,157.929
C02500=1047.574,362.377,379.913,173.314,41.083,157.931
C02501=1047.581,362.623,379.874,173.320,41.088,157.932
C02502=1047.589,362.870,379.836,173.325,41.092,157.933
C02503=1047.597,363.116,379.796,173.331,41.097,157.935
C02504=1047.605,363.364,379.758,173.335,41.101,157.936
C02505=1047.612,363.611,379.719,173.341,41.106,157.937
C02506=1047.620,363.857,379.680,173.347,41.111,157.939
C02507=1047.627,364.104,379.641,173.352,41.116,157.940
C02508=1047.635,364.351,379.602,173.358,41.120,157.942
C02509=1047.642,364.597,379.563,173.363,41.125,157.943
C02510=1047.650,364.845,379.524,173.369,41.130,157.945
C02511=1047.657,365.091,379.485,173.375,41.134,157.946
C02512=1047.666,365.338,379.446,173.380,41.140,157.948
C02513=1047.672,365.585,379.407,173.386,41.144,157.949
C02514=1047.680,365.832,379.367,173.392,41.149,157.950
C02515=1047.688,366.078,379.329,173.397,41.154,157.952
C02516=1047.695,366.325,379.289,173.403,41.158,157.953
C02517=1047.703,366.572,379.250,173.408,41.163,157.955
C02518=1047.711,366.819,379.211,173.415,41.168,157.956
C02519=1047.719,367.066,379.172,173.421,41.173,157.958
C02520=1047.726,367.313,379.132,173.426,41.177,157.959
C02521=1047.734,367.559,379.093,173.432,41.182,157.961
C02522=1047.742,367.806,379.054,173.438,41.187,157.962
C02523=1047.749,368.053,379.014,173.443,41.192,157.964
C02524=1047.757,368.299,378.975,173.449,41.197,157.965
C02525=1047.765,368.546,378.935,173.455,41.202,157.967
C02526=1047.773,368.793,378.897,173.460,41.207,157.968
C02527=1047.781,369.040,378.857,173.466,41.211,157.969
C02528=1047.789,369.286,378.818,173.472,41.217,157.971
C02529=1047.796,369.533,378.778,173.479,41.221,157.972
C02530=1047.804,369.780,378.738,173.484,41.226,157.974
C02531=1047.812,370.027,378.699,173.490,41.231,157.975
C02532=1047.819,370.273,378.660,173.496,41.236,157.977
C02533=1047.828,370.520,378.620,173.501,41.241,157.978
C02534=1047.836,370.767,378.580,173.507,41.246,157.980
C02535=1047.844,371.013,378.541,173.514,41.251,157.982
C02536=1047.852,371.260,378.501,173.520,41.256,157.983
C02537=1047.860,371.507,378.461,173.525,41.261,157.985
C02538=1047.867,371.753,378.421,173.531,41.266,157.986
C02539=1047.875,371.999,378.381,173.537,41.271,157.988
C02540=1047.882,372.246,378.341,173.543,41.276,157.989
C02541=1047.890,372.493,378.301,173.549,41.281,157.991
C02542=1047.899,372.740,378.262,173.555,41.286,157.992
C02543=1047.907,372.986,378.221,173.561,41.292,157.994
C02544=1047.914,373.233,378.181,173.567,41.297,157.996
C02545=1047.922,373.480,378.141,173.573,41.302,157.997
C02546=1047.929,373.726,378.101,173.580,41.307,157.999
C02547=1047.937,373.972,378.061,173.585,41.312,158.000
C02548=1047.945,374.219,378.021,173.591,41.318,158.002
C02549=1047.953,374.466,377.981,173.597,41.323,158.004
C02550=1047.961,374.713,377.941,173.604,41.328,158.005
C02551=1047.969,374.959,377.900,173.610,41.333,158.007
C02552=1047.980,375.292,377.846,173.618,41.340,158.009
C02553=1047.991,375.624,377.792,173.627,41.347,158.011
C02554=1048.001,375.957,377.738,173.634,41.354,158.013
C02555=1048.012,376.289,377.683,173.643,41.361,158.015
C02556=1048.020,376.535,377.643,173.650,41.367,158.017
C02557=1048.028,376.782,377.603,173.655,41.372,158.019
C02558=1048.036,377.028,377.562,173.661,41.377,158.020
C02559=1048.044,377.274,377.521,173.668,41.382,158.022
C02560=1048.051,377.521,377.482,173.674,41.388,158.024
C02561=1048.060,377.768,377.441,173.680,41.393,158.025
C02562=1048.068,378.015,377.400,173.687,41.398,158.027
C02563=1048.076,378.261,377.359,173.693,41.404,158.029
C02564=1048.084,378.507,377.319,173.699,41.409,158.030
C02565=1048.092,378.754,377.279,173.706,41.415,158.032
C02566=1048.100,379.001,377.238,173.712,41.420,158.034
C02567=1048.109,379.247,377.197,173.719,41.425,158.036
C02568=1048.117,379.493,377.157,173.724,41.431,158.037
C02569=1048.125,379.740,377.116,173.732,41.436,158.039
C02570=1048.133,379.987,377.075,173.737,41.441,158.040
C02571=1048.141,380.233,377.034,173.743,41.447,158.042
C02572=1048.149,380.479,376.992,173.750,41.453,158.044
C02573=1048.157,380.725,376.952,173.756,41.458,158.046
C02574=1048.165,380.972,376.911,173.763,41.463,158.047
C02575=1048.173,381.219,376.870,173.769,41.469,158.049
C02576=1048.181,381.465,376.829,173.776,41.475,158.051
C02577=1048.189,381.711,376.787,173.782,41.481,158.053
C02578=1048.198,381.958,376.746,173.790,41.486,158.054
C02579=1048.205,382.205,376.705,173.796,41.492,158.056
C02580=1048.213,382.450,376.664,173.803,41.497,158.058
C02581=1048.222,382.697,376.623,173.809,41.503,158.060
C02582=1048.230,382.944,376.582,173.816,41.509,158.062
C02583=1048.238,383.189,376.540,173.822,41.514,158.063
C02584=1048.246,383.436,376.499,173.829,41.520,158.065
C02585=1048.255,383.682,376.458,173.835,41.526,158.067
C02586=1048.262,383.929,376.416,173.842,41.531,158.069
C02587=1048.271,384.175,376.375,173.848,41.537,158.070
C02588=1048.279,384.422,376.334,173.855,41.543,158.072
C02589=1048.287,384.668,376.292,173.862,41.549,158.074
C02590=1048.295,384.914,376.251,173.868,41.554,158.076
C02591=1048.304,385.161,376.210,173.876,41.560,158.078
C02592=1048.312,385.407,376.167,173.882,41.566,158.079
C02593=1048.320,385.653,376.126,173.889,41.572,158.081
C02594=1048.329,385.900,376.085,173.896,41.577,158.083
C02595=1048.337,386.146,376.043,173.902,41.583,158.085
C02596=1048.346,386.392,376.001,173.909,41.589,158.087
C02597=1048.354,386.638,375.960,173.916,41.595,158.089
C02598=1048.362,386.885,375.918,173.923,41.601,158.091
C02599=1048.371,387.131,375.876,173.930,41.607,158.092
C02600=1048.379,387.377,375.834,173.937,41.613,158.094
C02601=1048.387,387.624,375.793,173.943,41.618,158.096
C02602=1048.396,387.870,375.751,173.950,41.625,158.098
C02603=1048.404,388.116,375.709,173.957,41.630,158.100
C02604=1048.413,388.363,375.668,173.964,41.636,158.102
C02605=1048.422,388.609,375.626,173.971,41.642,158.104
C02606=1048.430,388.856,375.584,173.978,41.648,158.106
C02607=1048.439,389.101,375.541,173.985,41.654,158.108
C02608=1048.451,389.467,375.479,173.996,41.663,158.110
C02609=1048.463,389.832,375.417,174.006,41.672,158.113
C02610=1048.476,390.197,375.354,174.016,41.681,158.116
C02611=1048.488,390.563,375.291,174.027,41.690,158.119
C02612=1048.497,390.809,375.248,174.034,41.696,158.121
C02613=1048.505,391.055,375.206,174.041,41.702,158.123
C02614=1048.514,391.302,375.164,174.048,41.709,158.125
C02615=1048.523,391.548,375.122,174.055,41.715,158.127
C02616=1048.530,391.794,375.080,174.063,41.721,158.129
C02617=1048.539,392.040,375.037,174.070,41.728,158.131
C02618=1048.548,392.286,374.995,174.077,41.734,158.133
C02619=1048.556,392.532,374.952,174.085,41.740,158.135
C02620=1048.565,392.778,374.909,174.092,41.746,158.137
C02621=1048.573,393.025,374.867,174.098,41.753,158.139
C02622=1048.582,393.271,374.824,174.106,41.759,158.141
C02623=1048.591,393.517,374.781,174.113,41.765,158.143
C02624=1048.599,393.763,374.738,174.120,41.771,158.145
C02625=1048.608,394.009,374.696,174.128,41.778,158.147
C02626=1048.616,394.255,374.653,174.135,41.784,158.149
C02627=1048.625,394.501,374.610,174.143,41.791,158.151
C02628=1048.634,394.747,374.567,174.150,41.797,158.153
C02629=1048.642,394.993,374.524,174.158,41.803,158.155
C02630=1048.651,395.239,374.481,174.165,41.810,158.157
C02631=1048.659,395.485,374.438,174.173,41.816,158.160
C02632=1048.668,395.731,374.395,174.180,41.822,158.162
C02633=1048.676,395.977,374.352,174.188,41.829,158.164
C02634=1048.686,396.223,374.310,174.195,41.836,158.166
C02635=1048.694,396.469,374.267,174.203,41.842,158.168
C02636=1048.703,396.715,374.224,174.210,41.849,158.170
C02637=1048.712,396.961,374.180,174.218,41.855,158.172
C02638=1048.720,397.207,374.136,174.225,41.862,158.174
C02639=1048.729,397.453,374.093,174.233,41.869,158.176
C02640=1048.738,397.699,374.050,174.240,41.875,158.179
C02641=1048.746,397.945,374.006,174.248,41.882,158.181
C02642=1048.755,398.192,373.963,174.255,41.888,158.183
C02643=1048.763,398.437,373.919,174.263,41.896,158.185
C02644=1048.772,398.684,373.876,174.272,41.902,158.187
C02645=1048.781,398.929,373.832,174.279,41.908,158.189
C02646=1048.790,399.176,373.789,174.287,41.915,158.192
C02647=1048.799,399.421,373.745,174.295,41.922,158.194
C02648=1048.807,399.667,373.702,174.302,41.929,158.196
C02649=1048.817,399.913,373.658,174.310,41.935,158.198
C02650=1048.825,400.159,373.615,174.317,41.942,158.200
C02651=1048.834,400.406,373.571,174.326,41.949,158.203
C02652=1048.843,400.651,373.527,174.334,41.956,158.205
C02653=1048.852,400.898,373.484,174.342,41.963,158.207
C02654=1048.861,401.143,373.440,174.349,41.970,158.209
C02655=1048.870,401.389,373.396,174.357,41.977,158.212
C02656=1048.879,401.635,373.351,174.366,41.984,158.214
C02657=1048.887,401.880,373.308,174.373,41.990,158.216
C02658=1048.897,402.127,373.264,174.381,41.997,158.218
C02659=1048.906,402.372,373.220,174.389,42.004,158.221
C02660=1048.914,402.618,373.175,174.398,42.011,158.223
C02661=1048.924,402.865,373.131,174.405,42.018,158.225
C02662=1048.933,403.110,373.087,174.413,42.026,158.228
C02663=1048.942,403.356,373.043,174.422,42.032,158.230
C02664=1048.950,403.602,372.999,174.430,42.040,158.232
C02665=1048.959,403.847,372.955,174.438,42.047,158.235
C02666=1048.969,404.093,372.910,174.446,42.054,158.237
C02667=1048.977,404.338,372.867,174.454,42.061,158.239
C02668=1048.987,404.584,372.822,174.462,42.068,158.242
C02669=1048.995,404.830,372.777,174.471,42.075,158.244
C02670=1049.004,405.074,372.733,174.479,42.082,158.246
C02671=1049.013,405.321,372.688,174.487,42.090,158.249
C02672=1049.023,405.566,372.643,174.496,42.097,158.251
C02673=1049.031,405.812,372.599,174.504,42.104,158.254
C02674=1049.040,406.058,372.554,174.512,42.111,158.256
C02675=1049.049,406.304,372.510,174.520,42.119,158.259
C02676=1049.059,406.550,372.465,174.529,42.126,158.261
C02677=1049.067,406.795,372.420,174.537,42.133,158.263
C02678=1049.077,407.041,372.376,174.546,42.141,158.266
C02679=1049.086,407.287,372.330,174.554,42.148,158.268
C02680=1049.095,407.533,372.286,174.563,42.155,158.271
C02681=1049.104,407.779,372.241,174.571,42.163,158.273
C02682=1049.114,408.024,372.196,174.580,42.170,158.276
C02683=1049.123,408.270,372.150,174.588,42.178,158.278
C02684=1049.132,408.515,372.106,174.597,42.185,158.281
C02685=1049.141,408.762,372.061,174.605,42.193,158.283
C02686=1049.151,409.007,372.016,174.614,42.200,158.286
C02687=1049.160,409.253,371.971,174.623,42.208,158.288
C02688=1049.169,409.499,371.925,174.632,42.215,158.291
C02689=1049.178,409.745,371.880,174.641,42.223,158.293
C02690=1049.187,409.990,371.835,174.650,42.231,158.296
C02691=1049.197,410.235,371.789,174.658,42.238,158.298
C02692=1049.206,410.481,371.744,174.667,42.246,158.301
C02693=1049.216,410.727,371.699,174.676,42.254,158.304
C02694=1049.226,410.973,371.653,174.684,42.261,158.306
C02695=1049.235,411.219,371.608,174.694,42.269,158.309
C02696=1049.245,411.464,371.562,174.703,42.276,158.311
C02697=1049.254,411.710,371.517,174.712,42.284,158.314
C02698=1049.263,411.955,371.472,174.720,42.292,158.317
C02699=1049.273,412.201,371.426,174.729,42.300,158.319
C02700=1049.282,412.447,371.380,174.739,42.308,158.322
C02701=1049.292,412.692,371.335,174.748,42.316,158.325
C02702=1049.302,412.938,371.289,174.757,42.323,158.327
C02703=1049.311,413.184,371.244,174.765,42.331,158.330
C02704=1049.326,413.568,371.172,174.781,42.343,158.334
C02705=1049.341,413.953,371.100,174.795,42.356,158.338
C02706=1049.356,414.336,371.028,174.809,42.369,158.343
C02707=1049.370,414.721,370.955,174.823,42.381,158.347
C02708=1049.381,414.967,370.909,174.833,42.390,158.350
C02709=1049.390,415.212,370.863,174.842,42.397,158.352
C02710=1049.400,415.458,370.817,174.851,42.405,158.355
C02711=1049.409,415.703,370.771,174.861,42.414,158.358
C02712=1049.419,415.949,370.724,174.870,42.422,158.361
C02713=1049.428,416.194,370.678,174.880,42.430,158.364
C02714=1049.438,416.439,370.631,174.889,42.438,158.367
C02715=1049.448,416.685,370.585,174.899,42.446,158.369
C02716=1049.458,416.930,370.538,174.908,42.455,158.372
C02717=1049.467,417.176,370.492,174.918,42.463,158.375
C02718=1049.477,417.422,370.446,174.927,42.472,158.378
C02719=1049.487,417.667,370.398,174.938,42.479,158.381
C02720=1049.503,418.058,370.324,174.953,42.493,158.385
C02721=1049.518,418.449,370.250,174.968,42.506,158.390
C02722=1049.534,418.840,370.175,174.984,42.520,158.395
C02723=1049.550,419.231,370.101,175.000,42.533,158.399
C02724=1049.560,419.476,370.054,175.010,42.542,158.402
C02725=1049.569,419.721,370.007,175.019,42.550,158.405
C02726=1049.579,419.967,369.960,175.030,42.559,158.408
C02727=1049.589,420.212,369.912,175.040,42.567,158.411
C02728=1049.600,420.457,369.865,175.049,42.576,158.414
C02729=1049.609,420.703,369.817,175.060,42.584,158.417
C02730=1049.619,420.948,369.770,175.070,42.593,158.420
C02731=1049.628,421.193,369.724,175.080,42.602,158.423
C02732=1049.639,421.438,369.676,175.091,42.611,158.426
C02733=1049.649,421.683,369.629,175.100,42.619,158.429
C02734=1049.659,421.929,369.581,175.110,42.628,158.432
C02735=1049.669,422.174,369.534,175.121,42.637,158.435
C02736=1049.679,422.419,369.487,175.131,42.646,158.438
C02737=1049.689,422.665,369.439,175.142,42.654,158.441
C02738=1049.699,422.911,369.391,175.152,42.664,158.445
C02739=1049.710,423.156,369.343,175.163,42.672,158.448
C02740=1049.720,423.401,369.296,175.172,42.681,158.451
C02741=1049.730,423.646,369.248,175.183,42.690,158.454
C02742=1049.740,423.891,369.200,175.193,42.699,158.457
C02743=1049.750,424.137,369.153,175.204,42.708,158.460
C02744=1049.761,424.381,369.105,175.215,42.717,158.464
C02745=1049.771,424.627,369.056,175.225,42.726,158.467
C02746=1049.781,424.872,369.009,175.236,42.735,158.470
C02747=1049.792,425.117,368.961,175.246,42.744,158.473
C02748=1049.802,425.362,368.912,175.257,42.753,158.476
C02749=1049.812,425.608,368.865,175.268,42.762,158.480
C02750=1049.822,425.853,368.817,175.279,42.772,158.483
C02751=1049.832,426.097,368.769,175.290,42.781,158.486
C02752=1049.843,426.343,368.720,175.301,42.790,158.489
C02753=1049.853,426.588,368.672,175.312,42.799,158.493
C02754=1049.863,426.833,368.623,175.322,42.808,158.496
C02755=1049.874,427.078,368.575,175.333,42.818,158.499
C02756=1049.884,427.323,368.526,175.345,42.827,158.503
C02757=1049.895,427.568,368.478,175.356,42.836,158.506
C02758=1049.905,427.813,368.429,175.367,42.846,158.509
C02759=1049.916,428.058,368.381,175.378,42.855,158.513
C02760=1049.926,428.303,368.332,175.390,42.865,158.516
C02761=1049.937,428.548,368.283,175.400,42.875,158.520
C02762=1049.947,428.793,368.235,175.411,42.884,158.523
C02763=1049.958,429.038,368.186,175.423,42.893,158.526
C02764=1049.969,429.283,368.137,175.434,42.903,158.530
C02765=1049.979,429.528,368.088,175.445,42.913,158.533
C02766=1049.990,429.773,368.039,175.457,42.922,158.537
C02767=1050.001,430.018,367.989,175.468,42.932,158.540
C02768=1050.010,430.263,367.941,175.480,42.941,158.544
C02769=1050.021,430.508,367.891,175.492,42.951,158.547
C02770=1050.032,430.753,367.842,175.504,42.961,158.551
C02771=1050.043,430.997,367.793,175.515,42.971,158.554
C02772=1050.053,431.242,367.743,175.527,42.981,158.558
C02773=1050.064,431.487,367.694,175.538,42.990,158.562
C02774=1050.075,431.732,367.644,175.550,43.001,158.565
C02775=1050.086,431.977,367.595,175.561,43.010,158.569
C02776=1050.103,432.391,367.511,175.582,43.027,158.575
C02777=1050.122,432.806,367.427,175.602,43.044,158.581
C02778=1050.140,433.219,367.344,175.622,43.061,158.587
C02779=1050.159,433.634,367.259,175.643,43.078,158.594
C02780=1050.170,433.878,367.209,175.655,43.088,158.597
C02781=1050.180,434.123,367.160,175.668,43.098,158.601
C02782=1050.191,434.368,367.109,175.680,43.108,158.605
C02783=1050.203,434.612,367.060,175.691,43.118,158.608
C02784=1050.214,434.858,367.010,175.704,43.129,158.612
C02785=1050.225,435.102,366.959,175.716,43.139,158.616
C02786=1050.236,435.347,366.910,175.729,43.149,158.620
C02787=1050.247,435.592,366.859,175.742,43.160,158.624
C02788=1050.258,435.836,366.809,175.754,43.170,158.628
C02789=1050.270,436.081,366.758,175.767,43.180,158.631
C02790=1050.281,436.325,366.709,175.779,43.191,158.635
C02791=1050.293,436.570,366.658,175.792,43.201,158.639
C02792=1050.304,436.815,366.608,175.805,43.212,158.643
C02793=1050.315,437.059,366.557,175.817,43.222,158.647
C02794=1050.325,437.304,366.506,175.830,43.233,158.651
C02795=1050.337,437.548,366.455,175.843,43.244,158.655
C02796=1050.348,437.793,366.405,175.856,43.254,158.659
C02797=1050.359,438.038,366.354,175.868,43.265,158.663
C02798=1050.371,438.282,366.303,175.882,43.275,158.667
C02799=1050.382,438.527,366.252,175.895,43.286,158.671
C02800=1050.394,438.771,366.201,175.908,43.297,158.675
C02801=1050.405,439.016,366.150,175.921,43.308,158.679
C02802=1050.416,439.260,366.099,175.935,43.318,158.683
C02803=1050.428,439.504,366.048,175.948,43.329,158.687
C02804=1050.439,439.748,365.996,175.961,43.340,158.691
C02805=1050.450,439.993,365.946,175.975,43.351,158.695
C02806=1050.462,440.238,365.894,175.988,43.362,158.700
C02807=1050.474,440.482,365.843,176.001,43.373,158.704
C02808=1050.486,440.726,365.792,176.015,43.384,158.708
C02809=1050.497,440.971,365.740,176.028,43.395,158.712
C02810=1050.509,441.216,365.688,176.042,43.406,158.716
C02811=1050.520,441.459,365.637,176.055,43.418,158.721
C02812=1050.532,441.703,365.585,176.069,43.429,158.725
C02813=1050.544,441.948,365.534,176.084,43.440,158.729
C02814=1050.555,442.193,365.482,176.097,43.451,158.734
C02815=1050.567,442.437,365.430,176.111,43.462,158.738
C02816=1050.579,442.681,365.378,176.124,43.474,158.742
C02817=1050.591,442.925,365.326,176.139,43.485,158.747
C02818=1050.602,443.170,365.274,176.153,43.496,158.751
C02819=1050.615,443.414,365.222,176.167,43.508,158.755
C02820=1050.626,443.658,365.169,176.181,43.519,158.760
C02821=1050.638,443.902,365.118,176.195,43.531,158.764
C02822=1050.650,444.146,365.066,176.210,43.542,158.769
C02823=1050.662,444.390,365.013,176.224,43.554,158.773
C02824=1050.674,444.634,364.961,176.239,43.565,158.778
C02825=1050.685,444.879,364.908,176.253,43.577,158.782
C02826=1050.698,445.123,364.856,176.268,43.589,158.787
C02827=1050.710,445.367,364.804,176.283,43.600,158.791
C02828=1050.722,445.610,364.751,176.297,43.612,158.796
C02829=1050.734,445.853,364.699,176.312,43.623,158.800
C02830=1050.747,446.097,364.646,176.327,43.635,158.805
C02831=1050.759,446.341,364.594,176.341,43.647,158.809
C02832=1050.776,446.643,364.530,176.359,43.661,158.815
C02833=1050.794,446.946,364.467,176.378,43.675,158.821
C02834=1050.814,447.251,364.405,176.397,43.689,158.826
C02835=1050.834,447.554,364.343,176.416,43.703,158.832
C02836=1050.851,447.799,364.294,176.431,43.713,158.836
C02837=1050.869,448.043,364.247,176.446,43.724,158.840
C02838=1050.888,448.288,364.198,176.462,43.734,158.845
C02839=1050.907,448.532,364.151,176.477,43.744,158.849
C02840=1050.926,448.777,364.104,176.493,43.754,158.853
C02841=1050.948,449.022,364.058,176.508,43.764,158.857
C02842=1050.969,449.267,364.013,176.525,43.774,158.862
C02843=1050.992,449.512,363.968,176.540,43.784,158.866
C02844=1051.014,449.757,363.924,176.556,43.793,158.870
C02845=1051.037,450.003,363.879,176.572,43.802,158.874
C02846=1051.061,450.247,363.836,176.588,43.811,158.878
C02847=1051.087,450.493,363.793,176.604,43.821,158.882
C02848=1050.772,450.520,363.495,176.604,43.914,158.909
C02849=1050.747,450.274,363.537,176.588,43.905,158.905
C02850=1050.722,450.029,363.581,176.571,43.896,158.901
C02851=1050.698,449.784,363.624,176.556,43.886,158.897
C02852=1050.675,449.538,363.669,176.540,43.877,158.893
C02853=1050.653,449.293,363.714,176.524,43.868,158.889
C02854=1050.631,449.048,363.759,176.508,43.858,158.884
C02855=1050.611,448.804,363.805,176.493,43.849,158.880
C02856=1050.591,448.559,363.852,176.477,43.839,158.876
C02857=1050.571,448.314,363.899,176.461,43.828,158.872
C02858=1050.552,448.069,363.946,176.446,43.818,158.867
C02859=1050.535,447.825,363.995,176.430,43.807,158.863
C02860=1050.517,447.581,364.043,176.414,43.797,158.859
C02861=1050.498,447.296,364.101,176.396,43.784,158.854
C02862=1050.480,447.009,364.160,176.379,43.772,158.848
C02863=1050.462,446.725,364.219,176.362,43.758,158.843
C02864=1050.446,446.440,364.278,176.344,43.745,158.838
C02865=1050.432,446.196,364.330,176.329,43.734,158.833
C02866=1050.420,445.953,364.383,176.314,43.723,158.829
C02867=1050.408,445.710,364.435,176.300,43.711,158.824
C02868=1050.395,445.466,364.488,176.285,43.699,158.820
C02869=1050.383,445.222,364.540,176.270,43.687,158.815
C02870=1050.371,444.978,364.592,176.256,43.676,158.810
C02871=1050.359,444.734,364.645,176.241,43.664,158.806
C02872=1050.347,444.490,364.697,176.226,43.653,158.801
C02873=1050.335,444.246,364.749,176.212,43.641,158.797
C02874=1050.323,444.002,364.802,176.197,43.630,158.793
C02875=1050.311,443.758,364.854,176.183,43.619,158.788
C02876=1050.299,443.514,364.906,176.168,43.607,158.784
C02877=1050.288,443.269,364.958,176.155,43.596,158.779
C02878=1050.276,443.025,365.010,176.141,43.585,158.775
C02879=1050.263,442.781,365.062,176.126,43.573,158.770
C02880=1050.252,442.536,365.114,176.112,43.562,158.766
C02881=1050.240,442.293,365.166,176.099,43.551,158.762
C02882=1050.228,442.048,365.218,176.084,43.540,158.757
C02883=1050.217,441.804,365.271,176.070,43.528,158.753
C02884=1050.205,441.559,365.322,176.057,43.517,158.749
C02885=1050.193,441.315,365.373,176.043,43.506,158.745
C02886=1050.181,441.070,365.425,176.029,43.495,158.740
C02887=1050.170,440.826,365.476,176.015,43.484,158.736
C02888=1050.159,440.582,365.528,176.002,43.473,158.732
C02889=1050.147,440.337,365.579,175.988,43.462,158.728
C02890=1050.135,440.093,365.631,175.975,43.451,158.724
C02891=1050.124,439.849,365.682,175.961,43.440,158.719
C02892=1050.112,439.604,365.733,175.948,43.430,158.715
C02893=1050.100,439.360,365.784,175.935,43.419,158.711
C02894=1050.089,439.116,365.836,175.921,43.408,158.707
C02895=1050.078,438.871,365.887,175.908,43.397,158.703
C02896=1050.066,438.627,365.938,175.895,43.387,158.699
C02897=1050.055,438.382,365.989,175.881,43.376,158.695
C02898=1050.044,438.138,366.040,175.868,43.365,158.691
C02899=1050.032,437.893,366.090,175.855,43.355,158.687
C02900=1050.021,437.649,366.141,175.843,43.344,158.683
C02901=1050.009,437.404,366.192,175.829,43.333,158.679
C02902=1049.998,437.159,366.242,175.816,43.323,158.675
C02903=1049.987,436.915,366.293,175.803,43.313,158.671
C02904=1049.975,436.670,366.344,175.791,43.302,158.667
C02905=1049.964,436.426,366.394,175.778,43.292,158.663
C02906=1049.953,436.181,366.445,175.765,43.281,158.659
C02907=1049.942,435.936,366.495,175.753,43.271,158.655
C02908=1049.931,435.692,366.546,175.740,43.261,158.652
C02909=1049.920,435.448,366.596,175.727,43.250,158.648
C02910=1049.909,435.202,366.646,175.715,43.240,158.644
C02911=1049.897,434.958,366.696,175.702,43.230,158.640
C02912=1049.886,434.713,366.746,175.691,43.220,158.636
C02913=1049.875,434.469,366.796,175.678,43.209,158.632
C02914=1049.864,434.224,366.846,175.666,43.199,158.629
C02915=1049.853,433.979,366.896,175.653,43.189,158.625
C02916=1049.841,433.734,366.946,175.641,43.179,158.621
C02917=1049.833,433.526,366.989,175.631,43.171,158.618
C02918=1049.824,433.318,367.031,175.620,43.162,158.615
C02919=1049.814,433.110,367.073,175.610,43.154,158.612
C02920=1049.805,432.901,367.115,175.600,43.145,158.609
C02921=1049.795,432.693,367.158,175.590,43.136,158.605
C02922=1049.786,432.485,367.200,175.579,43.129,158.602
C02923=1049.777,432.277,367.242,175.569,43.120,158.599
C02924=1049.767,432.068,367.285,175.559,43.111,158.596
C02925=1049.757,431.824,367.334,175.547,43.102,158.593
C02926=1049.746,431.579,367.383,175.535,43.092,158.589
C02927=1049.735,431.334,367.432,175.523,43.082,158.585
C02928=1049.725,431.089,367.482,175.511,43.072,158.582
C02929=1049.714,430.844,367.532,175.500,43.062,158.578
C02930=1049.703,430.600,367.580,175.489,43.053,158.575
C02931=1049.693,430.355,367.630,175.477,43.043,158.571
C02932=1049.682,430.110,367.680,175.465,43.033,158.568
C02933=1049.672,429.865,367.728,175.454,43.024,158.564
C02934=1049.661,429.620,367.778,175.441,43.014,158.561
C02935=1049.650,429.375,367.827,175.430,43.004,158.557
C02936=1049.640,429.129,367.876,175.419,42.995,158.554
C02937=1049.629,428.885,367.924,175.407,42.986,158.550
C02938=1049.619,428.640,367.973,175.396,42.976,158.547
C02939=1049.608,428.396,368.022,175.385,42.967,158.544
C02940=1049.597,428.150,368.071,175.374,42.957,158.540
C02941=1049.588,427.905,368.119,175.363,42.948,158.537
C02942=1049.576,427.660,368.168,175.352,42.938,158.533
C02943=1049.566,427.415,368.217,175.340,42.929,158.530
C02944=1049.555,427.170,368.265,175.329,42.920,158.527
C02945=1049.546,426.925,368.314,175.318,42.911,158.523
C02946=1049.534,426.680,368.362,175.307,42.901,158.520
C02947=1049.525,426.435,368.410,175.296,42.892,158.517
C02948=1049.514,426.189,368.459,175.285,42.883,158.513
C02949=1049.504,425.944,368.507,175.274,42.874,158.510
C02950=1049.493,425.700,368.555,175.263,42.865,158.507
C02951=1049.483,425.454,368.604,175.253,42.856,158.504
C02952=1049.472,425.209,368.652,175.242,42.847,158.500
C02953=1049.462,424.964,368.699,175.231,42.838,158.497
C02954=1049.453,424.719,368.748,175.221,42.829,158.494
C02955=1049.441,424.474,368.796,175.210,42.820,158.491
C02956=1049.431,424.228,368.843,175.199,42.811,158.488
C02957=1049.421,423.984,368.891,175.189,42.802,158.484
C02958=1049.411,423.738,368.939,175.178,42.793,158.481
C02959=1049.400,423.493,368.987,175.167,42.784,158.478
C02960=1049.390,423.247,369.034,175.157,42.775,158.475
C02961=1049.380,423.003,369.082,175.146,42.766,158.472
C02962=1049.370,422.757,369.130,175.136,42.757,158.469
C02963=1049.360,422.512,369.177,175.125,42.749,158.465
C02964=1049.350,422.267,369.225,175.115,42.740,158.462
C02965=1049.339,422.022,369.273,175.104,42.731,158.459
C02966=1049.330,421.776,369.320,175.094,42.722,158.456
C02967=1049.320,421.531,369.368,175.084,42.713,158.453
C02968=1049.309,421.286,369.415,175.074,42.705,158.450
C02969=1049.299,421.041,369.462,175.064,42.696,158.447
C02970=1049.290,420.795,369.510,175.053,42.688,158.444
C02971=1049.280,420.550,369.557,175.043,42.679,158.441
C02972=1049.269,420.304,369.604,175.033,42.670,158.438
C02973=1049.259,420.059,369.652,175.023,42.662,158.435
C02974=1049.250,419.814,369.698,175.013,42.653,158.432
C02975=1049.240,419.568,369.745,175.003,42.645,158.429
C02976=1049.230,419.323,369.793,174.994,42.637,158.426
C02977=1049.214,418.930,369.868,174.978,42.623,158.421
C02978=1049.198,418.537,369.943,174.962,42.610,158.417
C02979=1049.183,418.144,370.018,174.946,42.596,158.412
C02980=1049.167,417.750,370.092,174.930,42.583,158.407
C02981=1049.157,417.505,370.139,174.921,42.575,158.405
C02982=1049.148,417.260,370.186,174.910,42.567,158.402
C02983=1049.138,417.014,370.232,174.901,42.558,158.399
C02984=1049.127,416.769,370.279,174.891,42.550,158.396
C02985=1049.117,416.524,370.325,174.882,42.542,158.393
C02986=1049.108,416.278,370.371,174.872,42.534,158.390
C02987=1049.098,416.033,370.418,174.863,42.526,158.388
C02988=1049.088,415.787,370.464,174.853,42.517,158.385
C02989=1049.078,415.541,370.511,174.844,42.510,158.382
C02990=1049.069,415.296,370.557,174.834,42.501,158.379
C02991=1049.059,415.050,370.603,174.825,42.493,158.376
C02992=1049.050,414.805,370.649,174.815,42.485,158.374
C02993=1049.041,414.559,370.695,174.806,42.478,158.371
C02994=1049.031,414.314,370.742,174.796,42.469,158.368
C02995=1049.022,414.068,370.788,174.787,42.461,158.365
C02996=1049.012,413.822,370.835,174.778,42.453,158.363
C02997=1049.002,413.577,370.879,174.768,42.445,158.360
C02998=1048.993,413.332,370.926,174.760,42.437,158.357
C02999=1048.983,413.086,370.972,174.751,42.429,158.355
C03000=1048.974,412.840,371.017,174.741,42.422,158.352
C03001=1048.965,412.595,371.064,174.732,42.414,158.349
C03002=1048.954,412.349,371.109,174.723,42.406,158.347
C03003=1048.945,412.103,371.155,174.714,42.398,158.344
C03004=1048.936,411.858,371.200,174.704,42.391,158.341
C03005=1048.926,411.611,371.245,174.696,42.383,158.339
C03006=1048.916,411.366,371.292,174.687,42.376,158.336
C03007=1048.907,411.121,371.336,174.678,42.368,158.333
C03008=1048.898,410.875,371.382,174.669,42.360,158.331
C03009=1048.888,410.629,371.428,174.660,42.353,158.328
C03010=1048.878,410.383,371.473,174.651,42.345,158.326
C03011=1048.869,410.138,371.519,174.642,42.337,158.323
C03012=1048.859,409.892,371.563,174.634,42.330,158.321
C03013=1048.850,409.646,371.609,174.625,42.322,158.318
C03014=1048.841,409.401,371.654,174.616,42.315,158.316
C03015=1048.832,409.155,371.699,174.607,42.307,158.313
C03016=1048.822,408.909,371.744,174.598,42.300,158.310
C03017=1048.813,408.664,371.789,174.589,42.292,158.308
C03018=1048.804,408.418,371.835,174.581,42.285,158.305
C03019=1048.794,408.172,371.880,174.572,42.278,158.303
C03020=1048.785,407.926,371.925,174.564,42.270,158.300
C03021=1048.776,407.680,371.969,174.555,42.263,158.298
C03022=1048.767,407.434,372.015,174.546,42.255,158.295
C03023=1048.757,407.189,372.059,174.538,42.248,158.293
C03024=1048.748,406.943,372.105,174.529,42.241,158.291
C03025=1048.739,406.697,372.149,174.521,42.233,158.288
C03026=1048.730,406.451,372.194,174.512,42.226,158.286
C03027=1048.721,406.206,372.239,174.504,42.219,158.283
C03028=1048.712,405.960,372.283,174.495,42.211,158.281
C03029=1048.702,405.714,372.328,174.487,42.204,158.278
C03030=1048.694,405.468,372.373,174.479,42.197,158.276
C03031=1048.685,405.223,372.417,174.470,42.190,158.273
C03032=1048.676,404.977,372.462,174.463,42.183,158.271
C03033=1048.662,404.590,372.532,174.449,42.171,158.267
C03034=1048.648,404.204,372.602,174.436,42.160,158.264
C03035=1048.633,403.819,372.671,174.423,42.149,158.260
C03036=1048.619,403.433,372.741,174.411,42.138,158.256
C03037=1048.610,403.176,372.787,174.402,42.131,158.254
C03038=1048.600,402.920,372.833,174.394,42.124,158.251
C03039=1048.592,402.675,372.877,174.386,42.116,158.249
C03040=1048.582,402.429,372.921,174.377,42.110,158.247
C03041=1048.574,402.183,372.965,174.369,42.102,158.244
C03042=1048.565,401.937,373.009,174.361,42.095,158.242
C03043=1048.556,401.691,373.053,174.353,42.089,158.240
C03044=1048.546,401.445,373.097,174.345,42.082,158.238
C03045=1048.538,401.200,373.141,174.337,42.075,158.235
C03046=1048.529,400.953,373.185,174.330,42.068,158.233
C03047=1048.520,400.708,373.229,174.321,42.061,158.231
C03048=1048.511,400.461,373.273,174.313,42.055,158.229
C03049=1048.502,400.216,373.316,174.305,42.048,158.226
C03050=1048.493,399.969,373.360,174.298,42.041,158.224
C03051=1048.484,399.723,373.403,174.290,42.034,158.222
C03052=1048.475,399.477,373.448,174.281,42.028,158.220
C03053=1048.466,399.231,373.491,174.274,42.021,158.218
C03054=1048.458,398.986,373.534,174.266,42.014,158.215
C03055=1048.448,398.739,373.578,174.259,42.007,158.213
C03056=1048.440,398.494,373.621,174.251,42.001,158.211
C03057=1048.431,398.247,373.665,174.243,41.994,158.209
C03058=1048.422,398.002,373.708,174.236,41.988,158.207
C03059=1048.413,397.755,373.752,174.227,41.981,158.205
C03060=1048.405,397.509,373.795,174.220,41.975,158.202
C03061=1048.396,397.264,373.838,174.212,41.968,158.200
C03062=1048.387,397.018,373.881,174.205,41.962,158.198
C03063=1048.379,396.772,373.924,174.197,41.955,158.196
C03064=1048.370,396.526,373.969,174.189,41.948,158.194
C03065=1048.361,396.280,374.012,174.182,41.942,158.192
C03066=1048.353,396.033,374.055,174.174,41.935,158.190
C03067=1048.344,395.787,374.098,174.167,41.929,158.188
C03068=1048.336,395.541,374.141,174.159,41.923,158.185
C03069=1048.327,395.295,374.184,174.152,41.916,158.183
C03070=1048.318,395.050,374.226,174.144,41.910,158.181
C03071=1048.309,394.804,374.269,174.137,41.903,158.179
C03072=1048.301,394.557,374.312,174.129,41.897,158.177
C03073=1048.292,394.311,374.355,174.122,41.891,158.175
C03074=1048.284,394.065,374.398,174.114,41.884,158.173
C03075=1048.275,393.820,374.441,174.107,41.878,158.171
C03076=1048.266,393.573,374.483,174.100,41.871,158.169
C03077=1048.258,393.327,374.526,174.092,41.865,158.167
C03078=1048.249,393.081,374.569,174.085,41.859,158.165
C03079=1048.241,392.835,374.612,174.077,41.853,158.163
C03080=1048.232,392.588,374.654,174.071,41.846,158.161
C03081=1048.223,392.342,374.697,174.064,41.840,158.159
C03082=1048.215,392.096,374.740,174.056,41.834,158.157
C03083=1048.207,391.850,374.782,174.049,41.828,158.155
C03084=1048.197,391.604,374.825,174.041,41.822,158.153
C03085=1048.189,391.357,374.867,174.034,41.816,158.151
C03086=1048.181,391.112,374.910,174.027,41.810,158.149
C03087=1048.172,390.868,374.951,174.020,41.803,158.147
C03088=1048.164,390.626,374.993,174.013,41.797,158.145
C03089=1048.155,390.383,375.034,174.006,41.792,158.143
C03090=1048.148,390.140,375.076,173.999,41.786,158.141
C03091=1048.139,389.898,375.118,173.992,41.779,158.139
C03092=1048.131,389.655,375.159,173.985,41.773,158.137
C03093=1048.123,389.413,375.200,173.978,41.768,158.135
C03094=1048.114,389.170,375.242,173.972,41.762,158.133
C03095=1048.106,388.924,375.285,173.964,41.755,158.131
C03096=1048.097,388.678,375.327,173.957,41.750,158.130
C03097=1048.089,388.431,375.369,173.950,41.744,158.128
C03098=1048.080,388.185,375.410,173.944,41.738,158.126
C03099=1048.072,387.939,375.452,173.936,41.732,158.124
C03100=1048.063,387.692,375.494,173.929,41.726,158.122
C03101=1048.055,387.447,375.536,173.922,41.720,158.120
C03102=1048.047,387.200,375.578,173.916,41.714,158.118
C03103=1048.038,386.954,375.620,173.909,41.709,158.116
C03104=1048.029,386.708,375.661,173.902,41.703,158.115
C03105=1048.021,386.461,375.703,173.895,41.697,158.113
C03106=1048.012,386.214,375.744,173.888,41.691,158.111
C03107=1048.004,385.969,375.786,173.881,41.685,158.109
C03108=1047.996,385.722,375.828,173.875,41.679,158.107
C03109=1047.988,385.476,375.869,173.868,41.674,158.105
C03110=1047.979,385.229,375.910,173.861,41.668,158.104
C03111=1047.971,384.983,375.952,173.854,41.662,158.102
C03112=1047.962,384.737,375.994,173.847,41.657,158.100
C03113=1047.954,384.491,376.035,173.840,41.651,158.098
C03114=1047.946,384.244,376.077,173.834,41.645,158.096
C03115=1047.938,383.998,376.118,173.827,41.640,158.095
C03116=1047.929,383.751,376.159,173.821,41.634,158.093
C03117=1047.922,383.506,376.201,173.814,41.628,158.091
C03118=1047.913,383.259,376.242,173.808,41.623,158.089
C03119=1047.905,383.012,376.283,173.801,41.617,158.087
C03120=1047.897,382.766,376.325,173.793,41.612,158.086
C03121=1047.889,382.519,376.366,173.787,41.606,158.084
C03122=1047.880,382.274,376.407,173.780,41.600,158.082
C03123=1047.873,382.026,376.449,173.774,41.595,158.080
C03124=1047.865,381.780,376.489,173.767,41.589,158.078
C03125=1047.856,381.534,376.531,173.761,41.583,158.077
C03126=1047.848,381.288,376.571,173.754,41.578,158.075
C03127=1047.840,381.041,376.613,173.748,41.573,158.073
C03128=1047.832,380.795,376.654,173.741,41.567,158.072
C03129=1047.824,380.549,376.695,173.735,41.561,158.070
C03130=1047.816,380.302,376.736,173.729,41.556,158.068
C03131=1047.808,380.055,376.777,173.722,41.550,158.066
C03132=1047.800,379.809,376.818,173.716,41.545,158.065
C03133=1047.792,379.563,376.858,173.709,41.540,158.063
C03134=1047.784,379.316,376.899,173.703,41.534,158.061
C03135=1047.775,379.069,376.940,173.696,41.529,158.060
C03136=1047.767,378.823,376.981,173.690,41.523,158.058
C03137=1047.759,378.577,377.021,173.683,41.518,158.056
C03138=1047.751,378.331,377.062,173.677,41.513,158.055
C03139=1047.743,378.084,377.103,173.671,41.507,158.053
C03140=1047.735,377.837,377.143,173.664,41.502,158.051
C03141=1047.727,377.590,377.183,173.659,41.497,158.050
C03142=1047.719,377.344,377.224,173.651,41.491,158.048
C03143=1047.711,377.098,377.265,173.646,41.486,158.046
C03144=1047.703,376.851,377.305,173.640,41.481,158.045
C03145=1047.695,376.605,377.345,173.633,41.476,158.043
C03146=1047.686,376.358,377.386,173.627,41.471,158.041
C03147=1047.676,376.023,377.440,173.618,41.464,158.039
C03148=1047.665,375.689,377.495,173.610,41.456,158.037
C03149=1047.654,375.355,377.550,173.601,41.449,158.035
C03150=1047.643,375.020,377.604,173.594,41.442,158.033
C03151=1047.635,374.774,377.645,173.587,41.437,158.031
C03152=1047.627,374.527,377.685,173.581,41.432,158.029
C03153=1047.619,374.281,377.726,173.575,41.427,158.028
C03154=1047.612,374.034,377.765,173.568,41.422,158.026
C03155=1047.604,373.788,377.806,173.563,41.417,158.024
C03156=1047.596,373.541,377.846,173.557,41.411,158.023
C03157=1047.589,373.294,377.886,173.551,41.406,158.021
C03158=1047.580,373.048,377.926,173.544,41.401,158.020
C03159=1047.572,372.801,377.966,173.538,41.396,158.018
C03160=1047.565,372.555,378.005,173.533,41.391,158.017
C03161=1047.557,372.308,378.045,173.527,41.386,158.015
C03162=1047.549,372.061,378.086,173.521,41.381,158.013
C03163=1047.541,371.814,378.126,173.514,41.376,158.012
C03164=1047.534,371.568,378.165,173.508,41.371,158.010
C03165=1047.526,371.321,378.205,173.503,41.366,158.009
C03166=1047.518,371.075,378.245,173.497,41.361,158.007
C03167=1047.510,370.828,378.285,173.491,41.356,158.006
C03168=1047.502,370.581,378.325,173.484,41.351,158.004
C03169=1047.494,370.334,378.364,173.479,41.346,158.003
C03170=1047.487,370.088,378.403,173.473,41.341,158.001
C03171=1047.478,369.842,378.443,173.467,41.336,158.000
C03172=1047.471,369.595,378.483,173.461,41.331,157.998
C03173=1047.463,369.348,378.523,173.456,41.327,157.997
C03174=1047.454,369.101,378.562,173.449,41.322,157.995
C03175=1047.448,368.854,378.601,173.443,41.317,157.994
C03176=1047.439,368.608,378.640,173.438,41.312,157.992
C03177=1047.431,368.361,378.680,173.432,41.307,157.991
C03178=1047.423,368.114,378.719,173.426,41.302,157.989
C03179=1047.416,367.867,378.758,173.420,41.298,157.988
C03180=1047.408,367.620,378.798,173.415,41.293,157.986
C03181=1047.400,367.374,378.837,173.409,41.288,157.985
C03182=1047.393,367.127,378.876,173.403,41.283,157.983
C03183=1047.385,366.880,378.916,173.398,41.278,157.982
C03184=1047.377,366.634,378.955,173.391,41.274,157.980
C03185=1047.369,366.387,378.994,173.385,41.269,157.979
C03186=1047.362,366.140,379.034,173.380,41.264,157.978
C03187=1047.354,365.893,379.072,173.374,41.260,157.976
C03188=1047.346,365.647,379.112,173.368,41.255,157.974
C03189=1047.338,365.399,379.150,173.363,41.250,157.973
C03190=1047.331,365.153,379.190,173.357,41.245,157.972
C03191=1047.323,364.906,379.229,173.352,41.240,157.970
C03192=1047.316,364.660,379.268,173.346,41.236,157.969
C03193=1047.308,364.412,379.307,173.340,41.231,157.967
C03194=1047.301,364.166,379.346,173.335,41.226,157.966
C03195=1047.293,363.919,379.386,173.329,41.222,157.964
C03196=1047.286,363.672,379.424,173.323,41.217,157.963
C03197=1047.278,363.425,379.463,173.318,41.212,157.962
C03198=1047.270,363.179,379.502,173.312,41.208,157.960
C03199=1047.263,362.931,379.541,173.307,41.204,157.959
C03200=1047.255,362.685,379.579,173.301,41.199,157.957
C03201=1047.247,362.438,379.618,173.295,41.194,157.956
C03202=1047.240,362.191,379.657,173.290,41.190,157.955
C03203=1047.230,361.876,379.706,173.283,41.184,157.953
C03204=1047.220,361.560,379.755,173.276,41.178,157.951
C03205=1047.210,361.246,379.805,173.269,41.172,157.949
C03206=1047.201,360.930,379.854,173.262,41.167,157.948
C03207=1047.194,360.684,379.892,173.256,41.162,157.946
C03208=1047.185,360.437,379.931,173.252,41.158,157.945
C03209=1047.179,360.190,379.969,173.246,41.153,157.944
C03210=1047.170,359.943,380.008,173.241,41.149,157.942
C03211=1047.163,359.696,380.046,173.235,41.144,157.941
C03212=1047.155,359.450,380.084,173.230,41.140,157.940
C03213=1047.147,359.202,380.122,173.224,41.135,157.938
C03214=1047.141,358.955,380.161,173.219,41.131,157.937
C03215=1047.133,358.708,380.199,173.213,41.126,157.935
C03216=1047.125,358.461,380.238,173.208,41.122,157.934
C03217=1047.117,358.215,380.276,173.203,41.118,157.933
C03218=1047.110,357.968,380.314,173.198,41.113,157.932
C03219=1047.103,357.721,380.352,173.192,41.109,157.930
C03220=1047.095,357.473,380.391,173.187,41.104,157.929
C03221=1047.088,357.226,380.429,173.181,41.100,157.928
C03222=1047.080,356.980,380.467,173.176,41.096,157.926
C03223=1047.073,356.733,380.505,173.172,41.092,157.925
C03224=1047.065,356.485,380.543,173.166,41.087,157.924
C03225=1047.057,356.239,380.581,173.161,41.083,157.922
C03226=1047.050,355.992,380.619,173.155,41.079,157.921
C03227=1047.043,355.745,380.656,173.150,41.075,157.920
C03228=1047.035,355.497,380.695,173.145,41.070,157.919
C03229=1047.028,355.250,380.733,173.140,41.066,157.917
C03230=1047.020,355.004,380.771,173.134,41.062,157.916
C03231=1047.013,354.757,380.808,173.129,41.057,157.915
C03232=1047.006,354.510,380.846,173.124,41.053,157.913
C03233=1046.998,354.263,380.884,173.119,41.049,157.912
C03234=1046.990,354.015,380.922,173.114,41.045,157.911
C03235=1046.983,353.768,380.960,173.108,41.041,157.910
C03236=1046.975,353.522,380.998,173.103,41.037,157.908
C03237=1046.968,353.274,381.035,173.098,41.032,157.907
C03238=1046.961,353.027,381.073,173.093,41.028,157.906
C03239=1046.954,352.780,381.110,173.088,41.024,157.905
C03240=1046.946,352.534,381.149,173.083,41.020,157.903
C03241=1046.938,352.287,381.186,173.078,41.015,157.902
C03242=1046.931,352.040,381.223,173.072,41.011,157.901
C03243=1046.924,351.793,381.261,173.067,41.007,157.900
C03244=1046.916,351.545,381.298,173.063,41.003,157.898
C03245=1046.909,351.298,381.336,173.057,40.999,157.897
C03246=1046.902,351.051,381.373,173.052,40.995,157.896
C03247=1046.895,350.804,381.411,173.048,40.991,157.895
C03248=1046.887,350.557,381.448,173.042,40.987,157.893
C03249=1046.880,350.310,381.486,173.037,40.982,157.892
C03250=1046.872,350.063,381.523,173.032,40.978,157.891
C03251=1046.865,349.816,381.560,173.027,40.975,157.890
C03252=1046.858,349.569,381.598,173.022,40.970,157.889
C03253=1046.850,349.321,381.635,173.017,40.966,157.887
C03254=1046.842,349.075,381.672,173.012,40.963,157.886
C03255=1046.835,348.828,381.710,173.007,40.958,157.885
C03256=1046.828,348.580,381.747,173.002,40.954,157.884
C03257=1046.820,348.333,381.784,172.997,40.950,157.883
C03258=1046.813,348.086,381.821,172.992,40.946,157.881
C03259=1046.804,347.776,381.868,172.986,40.941,157.880
C03260=1046.794,347.467,381.914,172.980,40.936,157.878
C03261=1046.786,347.157,381.960,172.974,40.931,157.877
C03262=1046.776,346.848,382.006,172.967,40.926,157.875
C03263=1046.769,346.601,382.044,172.963,40.923,157.874
C03264=1046.762,346.353,382.081,172.958,40.918,157.873
C03265=1046.755,346.106,382.118,172.953,40.915,157.872
C03266=1046.747,345.858,382.154,172.948,40.910,157.871
C03267=1046.741,345.612,382.192,172.944,40.907,157.870
C03268=1046.733,345.365,382.228,172.938,40.902,157.868
C03269=1046.726,345.117,382.265,172.933,40.899,157.867
C03270=1046.718,344.870,382.303,172.929,40.895,157.866
C03271=1046.711,344.623,382.339,172.924,40.891,157.865
C03272=1046.704,344.376,382.375,172.919,40.887,157.864
C03273=1046.696,344.129,382.412,172.914,40.883,157.863
C03274=1046.690,343.881,382.449,172.910,40.879,157.862
C03275=1046.682,343.634,382.486,172.905,40.876,157.860
C03276=1046.675,343.387,382.523,172.900,40.871,157.859
C03277=1046.668,343.140,382.559,172.895,40.868,157.858
C03278=1046.660,342.893,382.596,172.891,40.864,157.857
C03279=1046.654,342.646,382.633,172.886,40.860,157.856
C03280=1046.646,342.398,382.669,172.881,40.856,157.855
C03281=1046.639,342.150,382.706,172.876,40.852,157.854
C03282=1046.632,341.904,382.742,172.872,40.849,157.853
C03283=1046.624,341.657,382.779,172.867,40.845,157.851
C03284=1046.617,341.409,382.815,172.863,40.841,157.850
C03285=1046.610,341.162,382.852,172.857,40.838,157.849
C03286=1046.603,340.915,382.887,172.853,40.834,157.848
C03287=1046.596,340.667,382.924,172.848,40.830,157.847
C03288=1046.589,340.420,382.960,172.844,40.826,157.846
C03289=1046.581,340.173,382.996,172.838,40.822,157.845
C03290=1046.574,339.925,383.033,172.834,40.819,157.844
C03291=1046.567,339.678,383.069,172.829,40.815,157.843
C03292=1046.559,339.431,383.105,172.825,40.811,157.841
C03293=1046.552,339.183,383.142,172.820,40.808,157.840
C03294=1046.545,338.937,383.178,172.815,40.804,157.839
C03295=1046.538,338.689,383.214,172.811,40.800,157.838
C03296=1046.531,338.442,383.251,172.806,40.796,157.837
C03297=1046.524,338.195,383.287,172.802,40.793,157.836
C03298=1046.516,337.948,383.323,172.797,40.789,157.835
C03299=1046.510,337.700,383.359,172.793,40.786,157.834
C03300=1046.502,337.453,383.395,172.788,40.782,157.833
C03301=1046.495,337.205,383.431,172.783,40.778,157.832
C03302=1046.489,336.958,383.467,172.779,40.775,157.831
C03303=1046.481,336.711,383.503,172.774,40.771,157.830
C03304=1046.474,336.464,383.539,172.770,40.767,157.829
C03305=1046.467,336.216,383.575,172.766,40.764,157.827
C03306=1046.460,335.969,383.611,172.760,40.760,157.826
C03307=1046.453,335.721,383.647,172.756,40.757,157.825
C03308=1046.446,335.474,383.683,172.752,40.753,157.824
C03309=1046.438,335.227,383.719,172.747,40.749,157.823
C03310=1046.431,334.980,383.755,172.743,40.746,157.822
C03311=1046.424,334.732,383.790,172.738,40.742,157.821
C03312=1046.417,334.485,383.826,172.734,40.739,157.820
C03313=1046.410,334.238,383.861,172.729,40.735,157.819
C03314=1046.402,333.990,383.897,172.724,40.732,157.818
C03315=1046.394,333.676,383.943,172.719,40.727,157.817
C03316=1046.385,333.363,383.988,172.714,40.723,157.816
C03317=1046.376,333.050,384.033,172.708,40.718,157.814
C03318=1046.366,332.737,384.078,172.703,40.714,157.813
C03319=1046.360,332.489,384.114,172.698,40.710,157.812
C03320=1046.353,332.242,384.149,172.693,40.707,157.811
C03321=1046.345,331.995,384.185,172.689,40.703,157.810
C03322=1046.338,331.747,384.220,172.684,40.700,157.809
C03323=1046.331,331.501,384.256,172.680,40.696,157.808
C03324=1046.324,331.252,384.291,172.676,40.693,157.807
C03325=1046.317,331.005,384.327,172.672,40.689,157.806
C03326=1046.310,330.758,384.362,172.667,40.686,157.805
C03327=1046.303,330.510,384.398,172.663,40.682,157.804
C03328=1046.296,330.263,384.433,172.659,40.679,157.803
C03329=1046.289,330.016,384.468,172.654,40.676,157.802
C03330=1046.282,329.768,384.503,172.649,40.672,157.801
C03331=1046.275,329.521,384.539,172.645,40.669,157.800
C03332=1046.268,329.273,384.575,172.641,40.665,157.799
C03333=1046.261,329.026,384.610,172.636,40.662,157.798
C03334=1046.253,328.778,384.645,172.632,40.659,157.797
C03335=1046.246,328.531,384.680,172.628,40.655,157.796
C03336=1046.240,328.284,384.715,172.624,40.652,157.795
C03337=1046.232,328.036,384.749,172.619,40.648,157.794
C03338=1046.225,327.788,384.785,172.615,40.645,157.793
C03339=1046.218,327.541,384.820,172.611,40.642,157.792
C03340=1046.210,327.294,384.855,172.607,40.638,157.791
C03341=1046.204,327.047,384.890,172.602,40.635,157.790
C03342=1046.196,326.799,384.925,172.598,40.632,157.789
C03343=1046.189,326.551,384.959,172.594,40.629,157.788
C03344=1046.182,326.304,384.994,172.590,40.626,157.787
C03345=1046.175,326.056,385.029,172.586,40.622,157.786
C03346=1046.168,325.809,385.064,172.581,40.619,157.785
C03347=1046.160,325.561,385.099,172.577,40.615,157.784
C03348=1046.153,325.314,385.134,172.573,40.612,157.783
C03349=1046.147,325.066,385.168,172.569,40.609,157.783
C03350=1046.139,324.819,385.203,172.565,40.606,157.782
C03351=1046.132,324.572,385.238,172.560,40.603,157.781
C03352=1046.125,324.325,385.273,172.556,40.599,157.780
C03353=1046.118,324.077,385.307,172.552,40.596,157.779
C03354=1046.112,323.829,385.342,172.548,40.593,157.778
C03355=1046.104,323.582,385.377,172.544,40.589,157.777
C03356=1046.097,323.333,385.411,172.540,40.586,157.776
C03357=1046.090,323.086,385.446,172.535,40.583,157.775
C03358=1046.083,322.839,385.481,172.531,40.580,157.774
C03359=1046.076,322.591,385.515,172.527,40.577,157.773
C03360=1046.069,322.344,385.550,172.523,40.573,157.772
C03361=1046.062,322.096,385.585,172.519,40.570,157.771
C03362=1046.055,321.849,385.619,172.515,40.567,157.770
C03363=1046.048,321.602,385.654,172.511,40.564,157.769
C03364=1046.041,321.354,385.688,172.507,40.561,157.769
C03365=1046.034,321.107,385.723,172.502,40.557,157.768
C03366=1046.027,320.859,385.757,172.498,40.554,157.767
C03367=1046.020,320.612,385.792,172.494,40.551,157.766
C03368=1046.013,320.364,385.826,172.490,40.548,157.765
C03369=1046.006,320.116,385.861,172.486,40.545,157.764
C03370=1046.000,319.869,385.895,172.482,40.541,157.763
C03371=1045.991,319.551,385.940,172.477,40.537,157.762
C03372=1045.982,319.232,385.983,172.471,40.533,157.761
C03373=1045.973,318.914,386.028,172.466,40.529,157.760
C03374=1045.965,318.595,386.072,172.461,40.525,157.758
C03375=1045.957,318.348,386.106,172.457,40.521,157.757
C03376=1045.951,318.101,386.140,172.453,40.518,157.756
C03377=1045.944,317.853,386.174,172.449,40.516,157.756
C03378=1045.937,317.606,386.209,172.445,40.512,157.755
C03379=1045.930,317.358,386.243,172.441,40.509,157.754
C03380=1045.924,317.110,386.278,172.437,40.506,157.753
C03381=1045.916,316.862,386.312,172.433,40.503,157.752
C03382=1045.910,316.616,386.346,172.429,40.499,157.751
C03383=1045.903,316.368,386.380,172.425,40.496,157.750
C03384=1045.897,316.120,386.415,172.421,40.493,157.749
C03385=1045.889,315.872,386.448,172.417,40.490,157.749
C03386=1045.884,315.625,386.482,172.413,40.487,157.748
C03387=1045.876,315.378,386.517,172.409,40.484,157.747
C03388=1045.870,315.130,386.551,172.405,40.481,157.746
C03389=1045.862,314.882,386.585,172.401,40.477,157.745
C03390=1045.857,314.635,386.619,172.397,40.474,157.744
C03391=1045.849,314.388,386.653,172.394,40.472,157.743
C03392=1045.843,314.140,386.687,172.390,40.468,157.742
C03393=1045.836,313.893,386.721,172.386,40.465,157.741
C03394=1045.829,313.645,386.755,172.382,40.462,157.740
C03395=1045.823,313.397,386.789,172.378,40.459,157.740
C03396=1045.816,313.150,386.823,172.374,40.456,157.739
C03397=1045.810,312.902,386.857,172.370,40.453,157.738
C03398=1045.802,312.654,386.891,172.366,40.450,157.737
C03399=1045.796,312.407,386.924,172.362,40.447,157.736
C03400=1045.789,312.160,386.958,172.358,40.444,157.735
C03401=1045.781,311.912,386.992,172.354,40.441,157.735
C03402=1045.774,311.664,387.025,172.350,40.438,157.734
C03403=1045.768,311.417,387.059,172.347,40.435,157.733
C03404=1045.761,311.169,387.092,172.343,40.432,157.732
C03405=1045.753,310.921,387.126,172.339,40.429,157.731
C03406=1045.747,310.673,387.159,172.336,40.426,157.730
C03407=1045.740,310.426,387.193,172.332,40.423,157.730
C03408=1045.733,310.178,387.227,172.328,40.420,157.729
C03409=1045.725,309.930,387.259,172.324,40.417,157.728
C03410=1045.719,309.683,387.293,172.321,40.415,157.727
C03411=1045.711,309.436,387.326,172.317,40.411,157.726
C03412=1045.704,309.187,387.360,172.313,40.409,157.725
C03413=1045.698,308.940,387.393,172.309,40.405,157.724
C03414=1045.691,308.692,387.426,172.305,40.403,157.724
C03415=1045.684,308.445,387.460,172.301,40.400,157.723
C03416=1045.677,308.198,387.493,172.297,40.397,157.722
C03417=1045.670,307.949,387.526,172.293,40.394,157.721
C03418=1045.663,307.703,387.559,172.289,40.391,157.720
C03419=1045.656,307.454,387.592,172.286,40.388,157.720
C03420=1045.649,307.207,387.626,172.282,40.386,157.719
C03421=1045.643,306.959,387.659,172.279,40.382,157.718
C03422=1045.636,306.712,387.692,172.275,40.380,157.717
C03423=1045.629,306.464,387.726,172.271,40.376,157.716
C03424=1045.622,306.216,387.759,172.267,40.374,157.716
C03425=1045.616,305.969,387.792,172.264,40.371,157.715
C03426=1045.608,305.721,387.825,172.260,40.368,157.714
C03427=1045.600,305.407,387.867,172.256,40.365,157.713
C03428=1045.592,305.094,387.909,172.250,40.361,157.712
C03429=1045.582,304.780,387.951,172.245,40.357,157.711
C03430=1045.574,304.466,387.993,172.241,40.353,157.710
C03431=1045.567,304.219,388.026,172.237,40.351,157.709
C03432=1045.561,303.970,388.059,172.234,40.348,157.708
C03433=1045.554,303.723,388.091,172.230,40.345,157.707
C03434=1045.546,303.475,388.125,172.226,40.342,157.707
C03435=1045.540,303.228,388.158,172.223,40.339,157.706
C03436=1045.534,302.980,388.190,172.219,40.337,157.705
C03437=1045.527,302.732,388.224,172.215,40.333,157.704
C03438=1045.520,302.485,388.257,172.212,40.331,157.703
C03439=1045.513,302.237,388.290,172.208,40.328,157.703
C03440=1045.506,301.989,388.322,172.205,40.325,157.702
C03441=1045.500,301.742,388.355,172.201,40.322,157.701
C03442=1045.493,301.493,388.388,172.197,40.319,157.700
C03443=1045.487,301.246,388.421,172.193,40.317,157.699
C03444=1045.480,300.999,388.454,172.190,40.314,157.699
C03445=1045.473,300.751,388.487,172.187,40.310,157.698
C03446=1045.466,300.503,388.520,172.183,40.308,157.697
C03447=1045.460,300.256,388.552,172.179,40.305,157.696
C03448=1045.453,300.007,388.585,172.175,40.302,157.696
C03449=1045.447,299.760,388.618,172.172,40.299,157.695
C03450=1045.440,299.513,388.650,172.169,40.296,157.694
C03451=1045.433,299.264,388.683,172.165,40.294,157.693
C03452=1045.427,299.017,388.716,172.161,40.291,157.692
C03453=1045.420,298.769,388.749,172.158,40.288,157.692
C03454=1045.414,298.521,388.782,172.154,40.285,157.691
C03455=1045.406,298.274,388.814,172.150,40.282,157.690
C03456=1045.400,298.026,388.847,172.147,40.280,157.689
C03457=1045.394,297.778,388.880,172.144,40.277,157.688
C03458=1045.388,297.531,388.912,172.140,40.274,157.688
C03459=1045.381,297.282,388.946,172.136,40.271,157.687
C03460=1045.374,297.035,388.978,172.133,40.268,157.686
C03461=1045.368,296.787,389.010,172.130,40.265,157.685
C03462=1045.361,296.539,389.042,172.126,40.263,157.685
C03463=1045.355,296.292,389.075,172.123,40.260,157.684
C03464=1045.347,296.044,389.108,172.119,40.257,157.683
C03465=1045.341,295.796,389.140,172.115,40.255,157.682
C03466=1045.335,295.548,389.172,172.113,40.252,157.682
C03467=1045.328,295.301,389.205,172.109,40.249,157.681
C03468=1045.322,295.053,389.237,172.105,40.246,157.680
C03469=1045.314,294.805,389.270,172.101,40.244,157.679
C03470=1045.308,294.557,389.302,172.099,40.241,157.679
C03471=1045.301,294.310,389.334,172.095,40.238,157.678
C03472=1045.294,294.062,389.365,172.091,40.236,157.677
C03473=1045.288,293.814,389.398,172.088,40.233,157.676
C03474=1045.281,293.566,389.431,172.084,40.230,157.676
C03475=1045.275,293.318,389.463,172.081,40.227,157.675
C03476=1045.267,293.071,389.495,172.078,40.225,157.674
C03477=1045.261,292.823,389.526,172.074,40.222,157.673
C03478=1045.254,292.575,389.559,172.070,40.219,157.673
C03479=1045.247,292.327,389.591,172.067,40.216,157.672
C03480=1045.240,292.079,389.623,172.064,40.214,157.671
C03481=1045.234,291.831,389.655,172.060,40.211,157.670
C03482=1045.227,291.584,389.687,172.057,40.208,157.670
C03483=1045.219,291.286,389.726,172.052,40.205,157.669
C03484=1045.212,290.989,389.764,172.048,40.202,157.668
C03485=1045.203,290.691,389.803,172.044,40.199,157.667
C03486=1045.195,290.394,389.840,172.041,40.196,157.666
C03487=1045.189,290.146,389.872,172.037,40.193,157.665
C03488=1045.181,289.898,389.905,172.034,40.190,157.665
C03489=1045.175,289.650,389.936,172.030,40.188,157.664
C03490=1045.168,289.402,389.968,172.027,40.185,157.663
C03491=1045.162,289.155,390.000,172.024,40.183,157.663
C03492=1045.155,288.907,390.032,172.020,40.180,157.662
C03493=1045.148,288.659,390.063,172.017,40.177,157.661
C03494=1045.142,288.411,390.095,172.013,40.175,157.660
C03495=1045.135,288.163,390.128,172.010,40.172,157.660
C03496=1045.129,287.915,390.159,172.007,40.169,157.659
C03497=1045.122,287.668,390.190,172.003,40.167,157.658
C03498=1045.115,287.420,390.222,172.001,40.164,157.657
C03499=1045.109,287.172,390.255,171.997,40.161,157.657
C03500=1045.102,286.924,390.286,171.994,40.159,157.656
C03501=1045.095,286.676,390.317,171.990,40.157,157.655
C03502=1045.089,286.428,390.349,171.987,40.154,157.655
C03503=1045.082,286.180,390.380,171.984,40.151,157.654
C03504=1045.075,285.933,390.412,171.980,40.148,157.653
C03505=1045.068,285.685,390.443,171.977,40.146,157.653
C03506=1045.062,285.437,390.475,171.974,40.143,157.652
C03507=1045.055,285.189,390.506,171.970,40.141,157.651
C03508=1045.048,284.941,390.537,171.967,40.138,157.650
C03509=1045.042,284.693,390.569,171.963,40.136,157.650
C03510=1045.035,284.445,390.600,171.961,40.133,157.649
C03511=1045.028,284.197,390.632,171.957,40.131,157.648
C03512=1045.021,283.949,390.663,171.954,40.128,157.648
C03513=1045.015,283.701,390.695,171.951,40.125,157.647
C03514=1045.008,283.453,390.726,171.948,40.123,157.646
C03515=1045.001,283.206,390.758,171.944,40.120,157.645
C03516=1044.994,282.958,390.789,171.941,40.118,157.645
C03517=1044.988,282.710,390.820,171.938,40.115,157.644
C03518=1044.981,282.462,390.852,171.935,40.113,157.643
C03519=1044.974,282.214,390.883,171.931,40.110,157.643
C03520=1044.968,281.965,390.914,171.928,40.107,157.642
C03521=1044.961,281.718,390.945,171.925,40.105,157.641
C03522=1044.954,281.470,390.977,171.922,40.102,157.641
C03523=1044.948,281.222,391.008,171.918,40.100,157.640
C03524=1044.942,280.975,391.039,171.916,40.097,157.639
C03525=1044.935,280.727,391.071,171.912,40.095,157.639
C03526=1044.928,280.478,391.101,171.909,40.092,157.638
C03527=1044.922,280.230,391.133,171.906,40.090,157.637
C03528=1044.915,279.982,391.164,171.903,40.087,157.636
C03529=1044.908,279.734,391.196,171.899,40.084,157.636
C03530=1044.902,279.486,391.226,171.896,40.082,157.635
C03531=1044.896,279.239,391.258,171.893,40.079,157.634
C03532=1044.889,278.991,391.289,171.890,40.077,157.634
C03533=1044.883,278.742,391.320,171.886,40.074,157.633
C03534=1044.876,278.494,391.351,171.884,40.071,157.632
C03535=1044.869,278.246,391.383,171.880,40.069,157.632
C03536=1044.862,277.998,391.413,171.877,40.067,157.631
C03537=1044.856,277.751,391.444,171.874,40.064,157.630
C03538=1044.849,277.503,391.474,171.871,40.062,157.630
C03539=1044.842,277.217,391.511,171.867,40.059,157.629
C03540=1044.834,276.931,391.545,171.863,40.056,157.628
C03541=1044.826,276.646,391.581,171.859,40.053,157.627
C03542=1044.819,276.360,391.617,171.857,40.050,157.627
C03543=1044.812,276.112,391.648,171.853,40.048,157.626
C03544=1044.805,275.863,391.678,171.850,40.045,157.625
C03545=1044.798,275.615,391.710,171.847,40.043,157.625
C03546=1044.792,275.368,391.740,171.844,40.040,157.624
C03547=1044.786,275.120,391.772,171.841,40.038,157.623
C03548=1044.779,274.872,391.802,171.837,40.035,157.622
C03549=1044.772,274.624,391.833,171.835,40.033,157.622
C03550=1044.765,274.375,391.864,171.831,40.030,157.621
C03551=1044.760,274.127,391.894,171.828,40.028,157.621
C03552=1044.752,273.880,391.925,171.826,40.025,157.620
C03553=1044.746,273.631,391.956,171.822,40.023,157.619
C03554=1044.740,273.383,391.986,171.819,40.020,157.619
C03555=1044.732,273.136,392.017,171.816,40.018,157.618
C03556=1044.726,272.887,392.048,171.813,40.015,157.617
C03557=1044.719,272.639,392.078,171.810,40.013,157.617
C03558=1044.713,272.392,392.109,171.807,40.010,157.616
C03559=1044.706,272.143,392.140,171.804,40.008,157.615
C03560=1044.699,271.895,392.170,171.800,40.005,157.615
C03561=1044.693,271.647,392.200,171.798,40.003,157.614
C03562=1044.687,271.399,392.231,171.795,40.001,157.613
C03563=1044.679,271.151,392.262,171.791,39.998,157.613
C03564=1044.674,270.903,392.292,171.789,39.996,157.612
C03565=1044.667,270.655,392.322,171.786,39.993,157.611
C03566=1044.660,270.407,392.353,171.782,39.991,157.611
C03567=1044.654,270.159,392.383,171.780,39.989,157.610
C03568=1044.647,269.911,392.414,171.777,39.986,157.609
C03569=1044.640,269.663,392.444,171.773,39.984,157.609
C03570=1044.634,269.415,392.474,171.771,39.981,157.608
C03571=1044.627,269.167,392.505,171.767,39.979,157.607
C03572=1044.620,268.918,392.535,171.764,39.977,157.607
C03573=1044.614,268.671,392.565,171.762,39.974,157.606
C03574=1044.607,268.422,392.596,171.758,39.972,157.606
C03575=1044.600,268.174,392.626,171.755,39.969,157.605
C03576=1044.594,267.926,392.656,171.753,39.967,157.604
C03577=1044.587,267.678,392.686,171.750,39.964,157.604
C03578=1044.581,267.431,392.716,171.746,39.962,157.603
C03579=1044.574,267.182,392.747,171.744,39.959,157.602
C03580=1044.567,266.934,392.777,171.741,39.957,157.602
C03581=1044.561,266.686,392.807,171.737,39.954,157.601
C03582=1044.554,266.438,392.837,171.735,39.952,157.600
C03583=1044.548,266.190,392.867,171.732,39.950,157.600
C03584=1044.541,265.942,392.898,171.729,39.947,157.599
C03585=1044.534,265.694,392.928,171.726,39.945,157.598
C03586=1044.528,265.445,392.957,171.723,39.943,157.598
C03587=1044.521,265.197,392.988,171.720,39.940,157.597
C03588=1044.515,264.949,393.018,171.717,39.938,157.597
C03589=1044.508,264.701,393.048,171.714,39.936,157.596
C03590=1044.502,264.453,393.078,171.712,39.933,157.595
C03591=1044.495,264.205,393.108,171.708,39.931,157.595
C03592=1044.488,263.957,393.137,171.705,39.928,157.594
C03593=1044.482,263.709,393.168,171.703,39.926,157.593
C03594=1044.475,263.461,393.198,171.700,39.923,157.593
C03595=1044.467,263.179,393.232,171.696,39.921,157.592
C03596=1044.460,262.898,393.266,171.693,39.918,157.591
C03597=1044.453,262.616,393.300,171.690,39.915,157.591
C03598=1044.445,262.335,393.333,171.686,39.912,157.590
C03599=1044.439,262.088,393.363,171.684,39.910,157.589
C03600=1044.432,261.839,393.393,171.681,39.908,157.589
C03601=1044.425,261.591,393.423,171.677,39.906,157.588
C03602=1044.419,261.343,393.452,171.675,39.903,157.587
C03603=1044.411,261.094,393.482,171.672,39.901,157.587
C03604=1044.405,260.847,393.512,171.669,39.898,157.586
C03605=1044.398,260.598,393.541,171.666,39.896,157.586
C03606=1044.391,260.351,393.571,171.663,39.894,157.585
C03607=1044.385,260.102,393.600,171.661,39.892,157.584
C03608=1044.378,259.854,393.630,171.658,39.889,157.584
C03609=1044.371,259.605,393.659,171.654,39.887,157.583
C03610=1044.365,259.358,393.689,171.652,39.885,157.583
C03611=1044.358,259.109,393.718,171.649,39.882,157.582
C03612=1044.351,258.862,393.748,171.646,39.880,157.581
C03613=1044.344,258.613,393.778,171.643,39.878,157.581
C03614=1044.337,258.365,393.806,171.640,39.876,157.580
C03615=1044.330,258.117,393.836,171.638,39.873,157.580
C03616=1044.324,257.869,393.865,171.635,39.871,157.579
C03617=1044.317,257.620,393.895,171.632,39.868,157.578
C03618=1044.311,257.372,393.924,171.629,39.866,157.578
C03619=1044.304,257.124,393.953,171.626,39.864,157.577
C03620=1044.297,256.876,393.984,171.624,39.862,157.577
C03621=1044.291,256.628,394.013,171.621,39.859,157.576
C03622=1044.284,256.379,394.042,171.618,39.857,157.575
C03623=1044.277,256.131,394.072,171.615,39.855,157.575
C03624=1044.271,255.883,394.101,171.612,39.852,157.574
C03625=1044.264,255.634,394.130,171.610,39.850,157.573
C03626=1044.258,255.387,394.160,171.607,39.848,157.573
C03627=1044.251,255.138,394.189,171.604,39.845,157.572
C03628=1044.245,254.890,394.218,171.602,39.843,157.572
C03629=1044.238,254.642,394.247,171.598,39.841,157.571
C03630=1044.231,254.394,394.277,171.595,39.838,157.570
C03631=1044.224,254.146,394.306,171.593,39.836,157.570
C03632=1044.218,253.898,394.335,171.590,39.834,157.569
